LIN {X 0,Y 353.361,Z 397.331,A -85,B 0,C 180,E1 -13405.436,E2 -13405.436} C_VEL
LIN {X 0,Y 353.277,Z 398.793,A -85,B 0,C 180,E1 -13406.578,E2 -13406.578} C_VEL
LIN {X 0,Y 353.318,Z 399.819,A -85,B 0,C 180,E1 -13407.719,E2 -13407.719} C_VEL
LIN {X 0,Y 353.397,Z 400.451,A -85,B 0,C 180,E1 -13408.86,E2 -13408.86} C_VEL
LIN {X 0,Y 353.406,Z 400.682,A -85,B 0,C 180,E1 -13409.999,E2 -13409.999} C_VEL
LIN {X 0,Y 353.397,Z 400.492,A -85,B 0,C 180,E1 -13411.139,E2 -13411.139} C_VEL
LIN {X 0,Y 353.319,Z 399.871,A -85,B 0,C 180,E1 -13412.279,E2 -13412.279} C_VEL
LIN {X 0,Y 353.359,Z 397.445,A -85,B 0,C 180,E1 -13414.562,E2 -13414.562} C_VEL
LIN {X 0,Y 353.439,Z 394.728,A -85,B 0,C 180,E1 -13416.149,E2 -13416.149} C_VEL
LIN {X 0,Y 353.657,Z 390.472,A -85,B 0,C 180,E1 -13417.995,E2 -13417.995} C_VEL
LIN {X 0,Y 354.202,Z 384.355,A -85,B 0,C 180,E1 -13419.997,E2 -13419.997} C_VEL
LIN {X 0,Y 354.848,Z 377.661,A -85,B 0,C 180,E1 -13421.712,E2 -13421.712} C_VEL
LIN {X 0,Y 355.833,Z 369.395,A -85,B 0,C 180,E1 -13423.418,E2 -13423.418} C_VEL
LIN {X 0,Y 356.776,Z 360.995,A -85,B 0,C 180,E1 -13424.837,E2 -13424.837} C_VEL
LIN {X 0,Y 357.808,Z 350.724,A -85,B 0,C 180,E1 -13426.253,E2 -13426.253} C_VEL
LIN {X 0,Y 359.128,Z 339.216,A -85,B 0,C 180,E1 -13427.51,E2 -13427.51} C_VEL
LIN {X 0,Y 359.906,Z 331.464,A -85,B 0,C 180,E1 -13428.205,E2 -13428.205} C_VEL
LIN {X 0,Y 358.662,Z 318.046,A -85,B 0,C 180,E1 -13429.294,E2 -13429.294} C_VEL
LIN {X 0,Y 357.078,Z 305.317,A -85,B 0,C 180,E1 -13430.105,E2 -13430.105} C_VEL
LIN {X 0,Y 354.409,Z 291.71,A -85,B 0,C 180,E1 -13430.818,E2 -13430.818} C_VEL
LIN {X 0,Y 354.987,Z 283.892,A -85,B 0,C 180,E1 -13434.566,E2 -13434.566} C_VEL
LIN {X 0,Y 355.743,Z 276.367,A -85,B 0,C 180,E1 -13438.302,E2 -13438.302} C_VEL
LIN {X 0,Y 356.393,Z 270.304,A -85,B 0,C 180,E1 -13441.447,E2 -13441.447} C_VEL
LIN {X 0,Y 357.263,Z 264.127,A -85,B 0,C 180,E1 -13444.783,E2 -13444.783} C_VEL
LIN {X 0,Y 357.549,Z 260.512,A -85,B 0,C 180,E1 -13446.86,E2 -13446.86} C_VEL
LIN {X 0,Y 357.149,Z 257.096,A -85,B 0,C 180,E1 -13449.027,E2 -13449.027} C_VEL
LIN {X 0,Y 356.306,Z 252.564,A -85,B 0,C 180,E1 -13452.115,E2 -13452.115} C_VEL
LIN {X 0,Y 355.547,Z 248.244,A -85,B 0,C 180,E1 -13455.364,E2 -13455.364} C_VEL
LIN {X 0,Y 354.843,Z 244.322,A -85,B 0,C 180,E1 -13458.686,E2 -13458.686} C_VEL
LIN {X 0,Y 354.814,Z 244.292,A -85,B 0,C 180,E1 -13462.4,E2 -13462.4} C_VEL
LIN {X 0,Y 354.813,Z 244.289,A -85,B 0,C 180,E1 -13464.939,E2 -13464.939} C_VEL
LIN {X 0,Y 354.793,Z 244.291,A -85,B 0,C 180,E1 -13468.403,E2 -13468.403} C_VEL
LIN {X 0,Y 354.849,Z 244.285,A -85,B 0,C 180,E1 -13471.617,E2 -13471.617} C_VEL
LIN {X 0,Y 354.899,Z 244.28,A -85,B 0,C 180,E1 -13474.171,E2 -13474.171} C_VEL
LIN {X 0,Y 354.834,Z 244.284,A -85,B 0,C 180,E1 -13477.892,E2 -13477.892} C_VEL
LIN {X 0,Y 354.922,Z 244.272,A -85,B 0,C 180,E1 -13481.89,E2 -13481.89} C_VEL
LIN {X 0,Y 354.941,Z 244.274,A -85,B 0,C 180,E1 -13485.979,E2 -13485.979} C_VEL
LIN {X 0,Y 354.975,Z 244.268,A -85,B 0,C 180,E1 -13489.734,E2 -13489.734} C_VEL
LIN {X 0,Y 355.111,Z 244.251,A -85,B 0,C 180,E1 -13492.035,E2 -13492.035} C_VEL
LIN {X 0,Y 355.09,Z 244.255,A -85,B 0,C 180,E1 -13494.319,E2 -13494.319} C_VEL
LIN {X 0,Y 355.242,Z 244.233,A -85,B 0,C 180,E1 -13497.731,E2 -13497.731} C_VEL
LIN {X 0,Y 355.395,Z 244.216,A -85,B 0,C 180,E1 -13499.998,E2 -13499.998} C_VEL
LIN {X 0,Y 355.241,Z 244.237,A -85,B 0,C 180,E1 -13502.266,E2 -13502.266} C_VEL
LIN {X 0,Y 355.134,Z 244.251,A -85,B 0,C 180,E1 -13506.817,E2 -13506.817} C_VEL
LIN {X 0,Y 354.999,Z 244.267,A -85,B 0,C 180,E1 -13509.111,E2 -13509.111} C_VEL
LIN {X 0,Y 354.849,Z 244.536,A -85,B 0,C 180,E1 -13511.421,E2 -13511.421} C_VEL
LIN {X 0,Y 354.814,Z 246.447,A -85,B 0,C 180,E1 -13513.938,E2 -13513.938} C_VEL
LIN {X 0,Y 354.579,Z 249.631,A -85,B 0,C 180,E1 -13517.94,E2 -13517.94} C_VEL
LIN {X 0,Y 354.357,Z 252.351,A -85,B 0,C 180,E1 -13521.229,E2 -13521.229} C_VEL
LIN {X 0,Y 354.214,Z 255.232,A -85,B 0,C 180,E1 -13524.622,E2 -13524.622} C_VEL
LIN {X 0,Y 354.178,Z 256.697,A -85,B 0,C 180,E1 -13526.277,E2 -13526.277} C_VEL
LIN {X 0,Y 358.421,Z 270.256,A -85,B 0,C 180,E1 -13527.172,E2 -13527.172} C_VEL
LIN {X 0,Y 361.22,Z 281.692,A -85,B 0,C 180,E1 -13528.071,E2 -13528.071} C_VEL
LIN {X 0,Y 361.763,Z 284.829,A -85,B 0,C 180,E1 -13528.34,E2 -13528.34} C_VEL
LIN {X 0,Y 360.778,Z 296.521,A -85,B 0,C 180,E1 -13529.301,E2 -13529.301} C_VEL
LIN {X 0,Y 359.767,Z 306.717,A -85,B 0,C 180,E1 -13530.359,E2 -13530.359} C_VEL
LIN {X 0,Y 358.53,Z 317.659,A -85,B 0,C 180,E1 -13531.788,E2 -13531.788} C_VEL
LIN {X 0,Y 357.331,Z 327.575,A -85,B 0,C 180,E1 -13533.413,E2 -13533.413} C_VEL
LIN {X 0,Y 356.279,Z 335.9,A -85,B 0,C 180,E1 -13535.138,E2 -13535.138} C_VEL
LIN {X 0,Y 355.322,Z 343.05,A -85,B 0,C 180,E1 -13537.002,E2 -13537.002} C_VEL
LIN {X 0,Y 354.684,Z 347.883,A -85,B 0,C 180,E1 -13538.603,E2 -13538.603} C_VEL
LIN {X 0,Y 354.224,Z 351.564,A -85,B 0,C 180,E1 -13540.149,E2 -13540.149} C_VEL
LIN {X 0,Y 353.897,Z 354.416,A -85,B 0,C 180,E1 -13541.713,E2 -13541.713} C_VEL
LIN {X 0,Y 353.712,Z 355.764,A -85,B 0,C 180,E1 -13542.68,E2 -13542.68} C_VEL
LIN {X 0,Y 353.482,Z 357.354,A -85,B 0,C 180,E1 -13544.296,E2 -13544.296} C_VEL
LIN {X 0,Y 353.306,Z 358.133,A -85,B 0,C 180,E1 -13545.876,E2 -13545.876} C_VEL
LIN {X 0,Y 353.236,Z 358.111,A -85,B 0,C 180,E1 -13547.433,E2 -13547.433} C_VEL
LIN {X 0,Y 353.343,Z 357.276,A -85,B 0,C 180,E1 -13549.093,E2 -13549.093} C_VEL
LIN {X 0,Y 353.518,Z 355.488,A -85,B 0,C 180,E1 -13550.83,E2 -13550.83} C_VEL
LIN {X 0,Y 353.811,Z 352.642,A -85,B 0,C 180,E1 -13552.608,E2 -13552.608} C_VEL
LIN {X 0,Y 354.233,Z 348.577,A -85,B 0,C 180,E1 -13554.429,E2 -13554.429} C_VEL
LIN {X 0,Y 354.798,Z 343.019,A -85,B 0,C 180,E1 -13556.315,E2 -13556.315} C_VEL
LIN {X 0,Y 355.556,Z 335.815,A -85,B 0,C 180,E1 -13558.201,E2 -13558.201} C_VEL
LIN {X 0,Y 356.447,Z 327.335,A -85,B 0,C 180,E1 -13559.958,E2 -13559.958} C_VEL
LIN {X 0,Y 357.46,Z 317.879,A -85,B 0,C 180,E1 -13561.526,E2 -13561.526} C_VEL
LIN {X 0,Y 358.429,Z 307.732,A -85,B 0,C 180,E1 -13562.879,E2 -13562.879} C_VEL
LIN {X 0,Y 359.445,Z 296.584,A -85,B 0,C 180,E1 -13564.074,E2 -13564.074} C_VEL
LIN {X 0,Y 360.348,Z 284.915,A -85,B 0,C 180,E1 -13565.055,E2 -13565.055} C_VEL
LIN {X 0,Y 360.523,Z 282.568,A -85,B 0,C 180,E1 -13565.222,E2 -13565.222} C_VEL
LIN {X 0,Y 358.332,Z 271.377,A -85,B 0,C 180,E1 -13566.056,E2 -13566.056} C_VEL
LIN {X 0,Y 354.955,Z 258.671,A -85,B 0,C 180,E1 -13566.827,E2 -13566.827} C_VEL
LIN {X 0,Y 353.815,Z 254.351,A -85,B 0,C 180,E1 -13567.057,E2 -13567.057} C_VEL
LIN {X 0,Y 353.884,Z 251.226,A -85,B 0,C 180,E1 -13570.269,E2 -13570.269} C_VEL
LIN {X 0,Y 354.007,Z 248.917,A -85,B 0,C 180,E1 -13572.676,E2 -13572.676} C_VEL
LIN {X 0,Y 354.162,Z 245.343,A -85,B 0,C 180,E1 -13576.485,E2 -13576.485} C_VEL
LIN {X 0,Y 354.227,Z 244.505,A -85,B 0,C 180,E1 -13577.395,E2 -13577.395} C_VEL
LIN {X 0,Y 354.713,Z 244.299,A -85,B 0,C 180,E1 -13580.881,E2 -13580.881} C_VEL
LIN {X 0,Y 355.055,Z 244.259,A -85,B 0,C 180,E1 -13583.18,E2 -13583.18} C_VEL
LIN {X 0,Y 355.231,Z 244.236,A -85,B 0,C 180,E1 -13587.733,E2 -13587.733} C_VEL
LIN {X 0,Y 355.383,Z 244.215,A -85,B 0,C 180,E1 -13590.001,E2 -13590.001} C_VEL
LIN {X 0,Y 355.231,Z 244.233,A -85,B 0,C 180,E1 -13592.268,E2 -13592.268} C_VEL
LIN {X 0,Y 355.123,Z 244.249,A -85,B 0,C 180,E1 -13596.82,E2 -13596.82} C_VEL
LIN {X 0,Y 355.002,Z 244.267,A -85,B 0,C 180,E1 -13599.113,E2 -13599.113} C_VEL
LIN {X 0,Y 354.911,Z 244.275,A -85,B 0,C 180,E1 -13602.582,E2 -13602.582} C_VEL
LIN {X 0,Y 354.875,Z 244.278,A -85,B 0,C 180,E1 -13606.097,E2 -13606.097} C_VEL
LIN {X 0,Y 354.896,Z 244.276,A -85,B 0,C 180,E1 -13608.473,E2 -13608.473} C_VEL
LIN {X 0,Y 354.874,Z 244.278,A -85,B 0,C 180,E1 -13612.104,E2 -13612.104} C_VEL
LIN {X 0,Y 354.887,Z 244.276,A -85,B 0,C 180,E1 -13615.829,E2 -13615.829} C_VEL
LIN {X 0,Y 354.841,Z 244.282,A -85,B 0,C 180,E1 -13619.68,E2 -13619.68} C_VEL
LIN {X 0,Y 354.795,Z 244.288,A -85,B 0,C 180,E1 -13623.704,E2 -13623.704} C_VEL
LIN {X 0,Y 354.789,Z 244.292,A -85,B 0,C 180,E1 -13626.461,E2 -13626.461} C_VEL
LIN {X 0,Y 354.814,Z 244.285,A -85,B 0,C 180,E1 -13629.426,E2 -13629.426} C_VEL
LIN {X 0,Y 354.826,Z 244.284,A -85,B 0,C 180,E1 -13631.226,E2 -13631.226} C_VEL
LIN {X 0,Y 354.125,Z 244.375,A -85,B 0,C 180,E1 -13632.173,E2 -13632.173} C_VEL
LIN {X 0,Y 351.255,Z 244.729,A -85,B 0,C 180,E1 -13633.712,E2 -13633.712} C_VEL
LIN {X 0,Y 348.861,Z 245.029,A -85,B 0,C 180,E1 -13634.957,E2 -13634.957} C_VEL
LIN {X 0,Y 347.859,Z 245.152,A -85,B 0,C 180,E1 -13635.921,E2 -13635.921} C_VEL
LIN {X 0,Y 347.79,Z 245.161,A -85,B 0,C 180,E1 -13636.247,E2 -13636.247} C_VEL
LIN {X 0,Y 347.778,Z 245.165,A -85,B 0,C 180,E1 -13640.168,E2 -13640.168} C_VEL
LIN {X 0,Y 347.783,Z 245.165,A -85,B 0,C 180,E1 -13644.127,E2 -13644.127} C_VEL
LIN {X 0,Y 347.759,Z 245.169,A -85,B 0,C 180,E1 -13648.305,E2 -13648.305} C_VEL
LIN {X 0,Y 347.802,Z 245.159,A -85,B 0,C 180,E1 -13650.992,E2 -13650.992} C_VEL
LIN {X 0,Y 347.828,Z 245.156,A -85,B 0,C 180,E1 -13653.61,E2 -13653.61} C_VEL
LIN {X 0,Y 347.786,Z 245.166,A -85,B 0,C 180,E1 -13656.164,E2 -13656.164} C_VEL
LIN {X 0,Y 347.816,Z 245.161,A -85,B 0,C 180,E1 -13659.912,E2 -13659.912} C_VEL
LIN {X 0,Y 347.865,Z 245.154,A -85,B 0,C 180,E1 -13662.362,E2 -13662.362} C_VEL
LIN {X 0,Y 347.897,Z 245.152,A -85,B 0,C 180,E1 -13665.973,E2 -13665.973} C_VEL
LIN {X 0,Y 347.927,Z 245.145,A -85,B 0,C 180,E1 -13669.528,E2 -13669.528} C_VEL
LIN {X 0,Y 348.08,Z 245.124,A -85,B 0,C 180,E1 -13673.044,E2 -13673.044} C_VEL
LIN {X 0,Y 348.208,Z 245.113,A -85,B 0,C 180,E1 -13677.689,E2 -13677.689} C_VEL
LIN {X 0,Y 348.347,Z 245.094,A -85,B 0,C 180,E1 -13680.002,E2 -13680.002} C_VEL
LIN {X 0,Y 348.208,Z 245.109,A -85,B 0,C 180,E1 -13682.315,E2 -13682.315} C_VEL
LIN {X 0,Y 348.067,Z 245.126,A -85,B 0,C 180,E1 -13686.96,E2 -13686.96} C_VEL
LIN {X 0,Y 347.901,Z 245.146,A -85,B 0,C 180,E1 -13690.477,E2 -13690.477} C_VEL
LIN {X 0,Y 347.904,Z 245.147,A -85,B 0,C 180,E1 -13694.151,E2 -13694.151} C_VEL
LIN {X 0,Y 347.897,Z 245.147,A -85,B 0,C 180,E1 -13698.291,E2 -13698.291} C_VEL
LIN {X 0,Y 347.793,Z 245.163,A -85,B 0,C 180,E1 -13701.636,E2 -13701.636} C_VEL
LIN {X 0,Y 347.818,Z 245.16,A -85,B 0,C 180,E1 -13705.11,E2 -13705.11} C_VEL
LIN {X 0,Y 347.815,Z 245.159,A -85,B 0,C 180,E1 -13707.695,E2 -13707.695} C_VEL
LIN {X 0,Y 347.756,Z 245.164,A -85,B 0,C 180,E1 -13710.349,E2 -13710.349} C_VEL
LIN {X 0,Y 347.755,Z 245.164,A -85,B 0,C 180,E1 -13714.045,E2 -13714.045} C_VEL
LIN {X 0,Y 347.768,Z 245.167,A -85,B 0,C 180,E1 -13717.322,E2 -13717.322} C_VEL
LIN {X 0,Y 347.739,Z 245.169,A -85,B 0,C 180,E1 -13720.298,E2 -13720.298} C_VEL
LIN {X 0,Y 347.776,Z 245.188,A -85,B 0,C 180,E1 -13723.096,E2 -13723.096} C_VEL
LIN {X 0,Y 348.766,Z 250.707,A -85,B 0,C 180,E1 -13726.753,E2 -13726.753} C_VEL
LIN {X 0,Y 349.769,Z 255.89,A -85,B 0,C 180,E1 -13729.985,E2 -13729.985} C_VEL
LIN {X 0,Y 350.482,Z 261.02,A -85,B 0,C 180,E1 -13733.017,E2 -13733.017} C_VEL
LIN {X 0,Y 350.039,Z 266.11,A -85,B 0,C 180,E1 -13735.793,E2 -13735.793} C_VEL
LIN {X 0,Y 349.258,Z 272.455,A -85,B 0,C 180,E1 -13739.127,E2 -13739.127} C_VEL
LIN {X 0,Y 348.563,Z 279.107,A -85,B 0,C 180,E1 -13742.521,E2 -13742.521} C_VEL
LIN {X 0,Y 347.849,Z 286.426,A -85,B 0,C 180,E1 -13746.166,E2 -13746.166} C_VEL
LIN {X 0,Y 347.374,Z 292.917,A -85,B 0,C 180,E1 -13749.291,E2 -13749.291} C_VEL
LIN {X 0,Y 349.68,Z 306.543,A -85,B 0,C 180,E1 -13749.923,E2 -13749.923} C_VEL
LIN {X 0,Y 351.362,Z 319.394,A -85,B 0,C 180,E1 -13750.738,E2 -13750.738} C_VEL
LIN {X 0,Y 352.641,Z 331.31,A -85,B 0,C 180,E1 -13751.706,E2 -13751.706} C_VEL
LIN {X 0,Y 351.608,Z 342.057,A -85,B 0,C 180,E1 -13752.702,E2 -13752.702} C_VEL
LIN {X 0,Y 350.415,Z 353.068,A -85,B 0,C 180,E1 -13753.988,E2 -13753.988} C_VEL
LIN {X 0,Y 349.438,Z 362.972,A -85,B 0,C 180,E1 -13755.439,E2 -13755.439} C_VEL
LIN {X 0,Y 348.513,Z 371.083,A -85,B 0,C 180,E1 -13756.887,E2 -13756.887} C_VEL
LIN {X 0,Y 347.547,Z 379.047,A -85,B 0,C 180,E1 -13758.628,E2 -13758.628} C_VEL
LIN {X 0,Y 347.062,Z 384.449,A -85,B 0,C 180,E1 -13760.088,E2 -13760.088} C_VEL
LIN {X 0,Y 346.596,Z 389.732,A -85,B 0,C 180,E1 -13761.839,E2 -13761.839} C_VEL
LIN {X 0,Y 346.342,Z 394.426,A -85,B 0,C 180,E1 -13763.896,E2 -13763.896} C_VEL
LIN {X 0,Y 346.276,Z 396.866,A -85,B 0,C 180,E1 -13765.343,E2 -13765.343} C_VEL
LIN {X 0,Y 346.201,Z 398.344,A -85,B 0,C 180,E1 -13766.508,E2 -13766.508} C_VEL
LIN {X 0,Y 346.317,Z 400.016,A -85,B 0,C 180,E1 -13768.837,E2 -13768.837} C_VEL
LIN {X 0,Y 346.345,Z 400.255,A -85,B 0,C 180,E1 -13769.999,E2 -13769.999} C_VEL
LIN {X 0,Y 346.318,Z 400.077,A -85,B 0,C 180,E1 -13771.162,E2 -13771.162} C_VEL
LIN {X 0,Y 346.207,Z 398.452,A -85,B 0,C 180,E1 -13773.491,E2 -13773.491} C_VEL
LIN {X 0,Y 346.273,Z 397.045,A -85,B 0,C 180,E1 -13774.656,E2 -13774.656} C_VEL
LIN {X 0,Y 346.335,Z 394.684,A -85,B 0,C 180,E1 -13776.092,E2 -13776.092} C_VEL
LIN {X 0,Y 346.595,Z 390.1,A -85,B 0,C 180,E1 -13778.159,E2 -13778.159} C_VEL
LIN {X 0,Y 347.072,Z 384.988,A -85,B 0,C 180,E1 -13779.91,E2 -13779.91} C_VEL
LIN {X 0,Y 347.687,Z 378.594,A -85,B 0,C 180,E1 -13781.661,E2 -13781.661} C_VEL
LIN {X 0,Y 348.717,Z 370.636,A -85,B 0,C 180,E1 -13783.401,E2 -13783.401} C_VEL
LIN {X 0,Y 349.88,Z 360.769,A -85,B 0,C 180,E1 -13785.136,E2 -13785.136} C_VEL
LIN {X 0,Y 350.976,Z 350.569,A -85,B 0,C 180,E1 -13786.579,E2 -13786.579} C_VEL
LIN {X 0,Y 352.371,Z 339.126,A -85,B 0,C 180,E1 -13787.857,E2 -13787.857} C_VEL
LIN {X 0,Y 353.017,Z 331.463,A -85,B 0,C 180,E1 -13788.574,E2 -13788.574} C_VEL
LIN {X 0,Y 351.865,Z 318.429,A -85,B 0,C 180,E1 -13789.665,E2 -13789.665} C_VEL
LIN {X 0,Y 350.342,Z 305.957,A -85,B 0,C 180,E1 -13790.504,E2 -13790.504} C_VEL
LIN {X 0,Y 347.884,Z 293.833,A -85,B 0,C 180,E1 -13791.177,E2 -13791.177} C_VEL
LIN {X 0,Y 347.426,Z 291.28,A -85,B 0,C 180,E1 -13791.298,E2 -13791.298} C_VEL
LIN {X 0,Y 348.044,Z 283.59,A -85,B 0,C 180,E1 -13795.09,E2 -13795.09} C_VEL
LIN {X 0,Y 348.821,Z 276.111,A -85,B 0,C 180,E1 -13798.917,E2 -13798.917} C_VEL
LIN {X 0,Y 349.564,Z 269.643,A -85,B 0,C 180,E1 -13802.389,E2 -13802.389} C_VEL
LIN {X 0,Y 350.429,Z 263.99,A -85,B 0,C 180,E1 -13805.563,E2 -13805.563} C_VEL
LIN {X 0,Y 350.493,Z 260.48,A -85,B 0,C 180,E1 -13807.703,E2 -13807.703} C_VEL
LIN {X 0,Y 349.865,Z 256.648,A -85,B 0,C 180,E1 -13810.239,E2 -13810.239} C_VEL
LIN {X 0,Y 349.01,Z 252.127,A -85,B 0,C 180,E1 -13813.535,E2 -13813.535} C_VEL
LIN {X 0,Y 348.364,Z 248.203,A -85,B 0,C 180,E1 -13816.69,E2 -13816.69} C_VEL
LIN {X 0,Y 347.784,Z 245.166,A -85,B 0,C 180,E1 -13819.537,E2 -13819.537} C_VEL
LIN {X 0,Y 347.768,Z 245.169,A -85,B 0,C 180,E1 -13822.678,E2 -13822.678} C_VEL
LIN {X 0,Y 347.749,Z 245.172,A -85,B 0,C 180,E1 -13825.955,E2 -13825.955} C_VEL
LIN {X 0,Y 347.764,Z 245.168,A -85,B 0,C 180,E1 -13829.652,E2 -13829.652} C_VEL
LIN {X 0,Y 347.851,Z 245.157,A -85,B 0,C 180,E1 -13832.743,E2 -13832.743} C_VEL
LIN {X 0,Y 347.788,Z 245.164,A -85,B 0,C 180,E1 -13836.16,E2 -13836.16} C_VEL
LIN {X 0,Y 347.816,Z 245.156,A -85,B 0,C 180,E1 -13839.908,E2 -13839.908} C_VEL
LIN {X 0,Y 347.865,Z 245.15,A -85,B 0,C 180,E1 -13842.357,E2 -13842.357} C_VEL
LIN {X 0,Y 347.895,Z 245.151,A -85,B 0,C 180,E1 -13845.969,E2 -13845.969} C_VEL
LIN {X 0,Y 347.926,Z 245.145,A -85,B 0,C 180,E1 -13849.524,E2 -13849.524} C_VEL
LIN {X 0,Y 348.071,Z 245.127,A -85,B 0,C 180,E1 -13851.873,E2 -13851.873} C_VEL
LIN {X 0,Y 348.065,Z 245.129,A -85,B 0,C 180,E1 -13854.204,E2 -13854.204} C_VEL
LIN {X 0,Y 348.205,Z 245.11,A -85,B 0,C 180,E1 -13857.685,E2 -13857.685} C_VEL
LIN {X 0,Y 348.365,Z 245.092,A -85,B 0,C 180,E1 -13859.998,E2 -13859.998} C_VEL
LIN {X 0,Y 348.203,Z 245.113,A -85,B 0,C 180,E1 -13862.312,E2 -13862.312} C_VEL
LIN {X 0,Y 348.103,Z 245.127,A -85,B 0,C 180,E1 -13866.956,E2 -13866.956} C_VEL
LIN {X 0,Y 347.931,Z 245.148,A -85,B 0,C 180,E1 -13869.297,E2 -13869.297} C_VEL
LIN {X 0,Y 347.849,Z 245.161,A -85,B 0,C 180,E1 -13870.475,E2 -13870.475} C_VEL
LIN {X 0,Y 347.784,Z 247.675,A -85,B 0,C 180,E1 -13874.078,E2 -13874.078} C_VEL
LIN {X 0,Y 347.574,Z 250.449,A -85,B 0,C 180,E1 -13877.654,E2 -13877.654} C_VEL
LIN {X 0,Y 347.335,Z 253.534,A -85,B 0,C 180,E1 -13881.448,E2 -13881.448} C_VEL
LIN {X 0,Y 347.139,Z 256.657,A -85,B 0,C 180,E1 -13885.158,E2 -13885.158} C_VEL
LIN {X 0,Y 347.121,Z 257.163,A -85,B 0,C 180,E1 -13885.762,E2 -13885.762} C_VEL
LIN {X 0,Y 351.833,Z 271.894,A -85,B 0,C 180,E1 -13886.796,E2 -13886.796} C_VEL
LIN {X 0,Y 354.664,Z 283.756,A -85,B 0,C 180,E1 -13887.783,E2 -13887.783} C_VEL
LIN {X 0,Y 355.097,Z 285.746,A -85,B 0,C 180,E1 -13887.97,E2 -13887.97} C_VEL
LIN {X 0,Y 354.11,Z 297.116,A -85,B 0,C 180,E1 -13888.928,E2 -13888.928} C_VEL
LIN {X 0,Y 352.84,Z 308.832,A -85,B 0,C 180,E1 -13890.192,E2 -13890.192} C_VEL
LIN {X 0,Y 351.623,Z 319.419,A -85,B 0,C 180,E1 -13891.643,E2 -13891.643} C_VEL
LIN {X 0,Y 350.492,Z 328.125,A -85,B 0,C 180,E1 -13893.118,E2 -13893.118} C_VEL
LIN {X 0,Y 349.479,Z 335.78,A -85,B 0,C 180,E1 -13894.723,E2 -13894.723} C_VEL
LIN {X 0,Y 348.394,Z 343.338,A -85,B 0,C 180,E1 -13896.715,E2 -13896.715} C_VEL
LIN {X 0,Y 347.726,Z 348.23,A -85,B 0,C 180,E1 -13898.361,E2 -13898.361} C_VEL
LIN {X 0,Y 347.116,Z 352.84,A -85,B 0,C 180,E1 -13900.38,E2 -13900.38} C_VEL
LIN {X 0,Y 346.766,Z 355.458,A -85,B 0,C 180,E1 -13901.973,E2 -13901.973} C_VEL
LIN {X 0,Y 346.484,Z 357.303,A -85,B 0,C 180,E1 -13903.599,E2 -13903.599} C_VEL
LIN {X 0,Y 346.277,Z 358.373,A -85,B 0,C 180,E1 -13905.26,E2 -13905.26} C_VEL
LIN {X 0,Y 346.165,Z 358.629,A -85,B 0,C 180,E1 -13906.957,E2 -13906.957} C_VEL
LIN {X 0,Y 346.215,Z 358.016,A -85,B 0,C 180,E1 -13908.68,E2 -13908.68} C_VEL
LIN {X 0,Y 346.383,Z 356.463,A -85,B 0,C 180,E1 -13910.44,E2 -13910.44} C_VEL
LIN {X 0,Y 346.743,Z 353.31,A -85,B 0,C 180,E1 -13912.552,E2 -13912.552} C_VEL
LIN {X 0,Y 347.058,Z 350.115,A -85,B 0,C 180,E1 -13914.092,E2 -13914.092} C_VEL
LIN {X 0,Y 347.617,Z 344.953,A -85,B 0,C 180,E1 -13915.984,E2 -13915.984} C_VEL
LIN {X 0,Y 348.319,Z 338.108,A -85,B 0,C 180,E1 -13917.928,E2 -13917.928} C_VEL
LIN {X 0,Y 349.101,Z 331.426,A -85,B 0,C 180,E1 -13919.449,E2 -13919.449} C_VEL
LIN {X 0,Y 350.076,Z 322.94,A -85,B 0,C 180,E1 -13921.033,E2 -13921.033} C_VEL
LIN {X 0,Y 351.14,Z 312.518,A -85,B 0,C 180,E1 -13922.592,E2 -13922.592} C_VEL
LIN {X 0,Y 352.253,Z 301.01,A -85,B 0,C 180,E1 -13923.965,E2 -13923.965} C_VEL
LIN {X 0,Y 353.249,Z 289.115,A -85,B 0,C 180,E1 -13925.069,E2 -13925.069} C_VEL
LIN {X 0,Y 353.691,Z 283.577,A -85,B 0,C 180,E1 -13925.494,E2 -13925.494} C_VEL
LIN {X 0,Y 351.235,Z 271.767,A -85,B 0,C 180,E1 -13926.411,E2 -13926.411} C_VEL
LIN {X 0,Y 347.924,Z 259.115,A -85,B 0,C 180,E1 -13927.197,E2 -13927.197} C_VEL
LIN {X 0,Y 346.766,Z 254.748,A -85,B 0,C 180,E1 -13927.431,E2 -13927.431} C_VEL
LIN {X 0,Y 346.872,Z 251.238,A -85,B 0,C 180,E1 -13931.085,E2 -13931.085} C_VEL
LIN {X 0,Y 346.945,Z 248.94,A -85,B 0,C 180,E1 -13933.526,E2 -13933.526} C_VEL
LIN {X 0,Y 347.173,Z 245.603,A -85,B 0,C 180,E1 -13937.134,E2 -13937.134} C_VEL
LIN {X 0,Y 347.46,Z 245.207,A -85,B 0,C 180,E1 -13939.512,E2 -13939.512} C_VEL
LIN {X 0,Y 348.013,Z 245.135,A -85,B 0,C 180,E1 -13943.041,E2 -13943.041} C_VEL
LIN {X 0,Y 348.193,Z 245.112,A -85,B 0,C 180,E1 -13947.687,E2 -13947.687} C_VEL
LIN {X 0,Y 348.353,Z 245.09,A -85,B 0,C 180,E1 -13950.001,E2 -13950.001} C_VEL
LIN {X 0,Y 348.193,Z 245.11,A -85,B 0,C 180,E1 -13952.314,E2 -13952.314} C_VEL
LIN {X 0,Y 348.091,Z 245.127,A -85,B 0,C 180,E1 -13956.959,E2 -13956.959} C_VEL
LIN {X 0,Y 347.954,Z 245.144,A -85,B 0,C 180,E1 -13959.299,E2 -13959.299} C_VEL
LIN {X 0,Y 347.879,Z 245.153,A -85,B 0,C 180,E1 -13962.84,E2 -13962.84} C_VEL
LIN {X 0,Y 347.825,Z 245.157,A -85,B 0,C 180,E1 -13966.433,E2 -13966.433} C_VEL
LIN {X 0,Y 347.849,Z 245.158,A -85,B 0,C 180,E1 -13968.861,E2 -13968.861} C_VEL
LIN {X 0,Y 347.795,Z 245.162,A -85,B 0,C 180,E1 -13972.578,E2 -13972.578} C_VEL
LIN {X 0,Y 347.808,Z 245.161,A -85,B 0,C 180,E1 -13975.109,E2 -13975.109} C_VEL
LIN {X 0,Y 347.797,Z 245.159,A -85,B 0,C 180,E1 -13977.696,E2 -13977.696} C_VEL
LIN {X 0,Y 347.752,Z 245.167,A -85,B 0,C 180,E1 -13980.348,E2 -13980.348} C_VEL
LIN {X 0,Y 347.733,Z 245.171,A -85,B 0,C 180,E1 -13984.466,E2 -13984.466} C_VEL
LIN {X 0,Y 347.766,Z 245.164,A -85,B 0,C 180,E1 -13987.991,E2 -13987.991} C_VEL
LIN {X 0,Y 347.775,Z 245.162,A -85,B 0,C 180,E1 -13991.611,E2 -13991.611} C_VEL
LIN {X 0,Y 347.822,Z 245.158,A -85,B 0,C 180,E1 -13995.008,E2 -13995.008} C_VEL
LIN {X 0,Y 347.79,Z 245.161,A -85,B 0,C 180,E1 -13996.247,E2 -13996.247} C_VEL
LIN {X 0,Y 347.143,Z 245.247,A -85,B 0,C 180,E1 -13997.214,E2 -13997.214} C_VEL
LIN {X 0,Y 344.257,Z 245.605,A -85,B 0,C 180,E1 -13998.786,E2 -13998.786} C_VEL
LIN {X 0,Y 341.806,Z 245.908,A -85,B 0,C 180,E1 -14000.059,E2 -14000.059} C_VEL
LIN {X 0,Y 340.774,Z 246.035,A -85,B 0,C 180,E1 -14001.044,E2 -14001.044} C_VEL
LIN {X 0,Y 340.701,Z 246.042,A -85,B 0,C 180,E1 -14001.378,E2 -14001.378} C_VEL
LIN {X 0,Y 340.713,Z 246.044,A -85,B 0,C 180,E1 -14004.724,E2 -14004.724} C_VEL
LIN {X 0,Y 340.711,Z 246.042,A -85,B 0,C 180,E1 -14008.96,E2 -14008.96} C_VEL
LIN {X 0,Y 340.776,Z 246.037,A -85,B 0,C 180,E1 -14012.476,E2 -14012.476} C_VEL
LIN {X 0,Y 340.753,Z 246.038,A -85,B 0,C 180,E1 -14015.641,E2 -14015.641} C_VEL
LIN {X 0,Y 340.746,Z 246.038,A -85,B 0,C 180,E1 -14019.477,E2 -14019.477} C_VEL
LIN {X 0,Y 340.857,Z 246.029,A -85,B 0,C 180,E1 -14021.987,E2 -14021.987} C_VEL
LIN {X 0,Y 340.869,Z 246.025,A -85,B 0,C 180,E1 -14025.707,E2 -14025.707} C_VEL
LIN {X 0,Y 340.87,Z 246.023,A -85,B 0,C 180,E1 -14029.308,E2 -14029.308} C_VEL
LIN {X 0,Y 341.047,Z 246,A -85,B 0,C 180,E1 -14032.9,E2 -14032.9} C_VEL
LIN {X 0,Y 341.17,Z 245.989,A -85,B 0,C 180,E1 -14037.641,E2 -14037.641} C_VEL
LIN {X 0,Y 341.298,Z 245.972,A -85,B 0,C 180,E1 -14040.002,E2 -14040.002} C_VEL
LIN {X 0,Y 341.17,Z 245.985,A -85,B 0,C 180,E1 -14042.363,E2 -14042.363} C_VEL
LIN {X 0,Y 341.013,Z 246.005,A -85,B 0,C 180,E1 -14047.105,E2 -14047.105} C_VEL
LIN {X 0,Y 340.852,Z 246.024,A -85,B 0,C 180,E1 -14050.696,E2 -14050.696} C_VEL
LIN {X 0,Y 340.868,Z 246.022,A -85,B 0,C 180,E1 -14054.326,E2 -14054.326} C_VEL
LIN {X 0,Y 340.843,Z 246.025,A -85,B 0,C 180,E1 -14058.468,E2 -14058.468} C_VEL
LIN {X 0,Y 340.76,Z 246.037,A -85,B 0,C 180,E1 -14061.858,E2 -14061.858} C_VEL
LIN {X 0,Y 340.778,Z 246.036,A -85,B 0,C 180,E1 -14065.666,E2 -14065.666} C_VEL
LIN {X 0,Y 340.735,Z 246.039,A -85,B 0,C 180,E1 -14068.322,E2 -14068.322} C_VEL
LIN {X 0,Y 340.705,Z 246.046,A -85,B 0,C 180,E1 -14071.046,E2 -14071.046} C_VEL
LIN {X 0,Y 340.725,Z 246.045,A -85,B 0,C 180,E1 -14075.28,E2 -14075.28} C_VEL
LIN {X 0,Y 340.717,Z 246.045,A -85,B 0,C 180,E1 -14078.387,E2 -14078.387} C_VEL
LIN {X 0,Y 340.732,Z 246.04,A -85,B 0,C 180,E1 -14082.421,E2 -14082.421} C_VEL
LIN {X 0,Y 340.77,Z 246.34,A -85,B 0,C 180,E1 -14082.891,E2 -14082.891} C_VEL
LIN {X 0,Y 341.624,Z 250.986,A -85,B 0,C 180,E1 -14086.059,E2 -14086.059} C_VEL
LIN {X 0,Y 342.6,Z 256.138,A -85,B 0,C 180,E1 -14089.379,E2 -14089.379} C_VEL
LIN {X 0,Y 343.312,Z 260.621,A -85,B 0,C 180,E1 -14092.11,E2 -14092.11} C_VEL
LIN {X 0,Y 343.413,Z 263.171,A -85,B 0,C 180,E1 -14093.594,E2 -14093.594} C_VEL
LIN {X 0,Y 342.894,Z 268.273,A -85,B 0,C 180,E1 -14096.399,E2 -14096.399} C_VEL
LIN {X 0,Y 342.091,Z 274.323,A -85,B 0,C 180,E1 -14099.641,E2 -14099.641} C_VEL
LIN {X 0,Y 341.365,Z 280.939,A -85,B 0,C 180,E1 -14103.067,E2 -14103.067} C_VEL
LIN {X 0,Y 340.761,Z 287.25,A -85,B 0,C 180,E1 -14106.285,E2 -14106.285} C_VEL
LIN {X 0,Y 340.357,Z 292.422,A -85,B 0,C 180,E1 -14108.866,E2 -14108.866} C_VEL
LIN {X 0,Y 342.895,Z 307.742,A -85,B 0,C 180,E1 -14109.635,E2 -14109.635} C_VEL
LIN {X 0,Y 344.454,Z 319.682,A -85,B 0,C 180,E1 -14110.43,E2 -14110.43} C_VEL
LIN {X 0,Y 345.729,Z 332.17,A -85,B 0,C 180,E1 -14111.48,E2 -14111.48} C_VEL
LIN {X 0,Y 344.484,Z 343.953,A -85,B 0,C 180,E1 -14112.64,E2 -14112.64} C_VEL
LIN {X 0,Y 343.316,Z 354.54,A -85,B 0,C 180,E1 -14113.957,E2 -14113.957} C_VEL
LIN {X 0,Y 342.312,Z 364.116,A -85,B 0,C 180,E1 -14115.433,E2 -14115.433} C_VEL
LIN {X 0,Y 341.169,Z 373.336,A -85,B 0,C 180,E1 -14117.205,E2 -14117.205} C_VEL
LIN {X 0,Y 340.329,Z 380.762,A -85,B 0,C 180,E1 -14118.987,E2 -14118.987} C_VEL
LIN {X 0,Y 339.703,Z 387.596,A -85,B 0,C 180,E1 -14121.073,E2 -14121.073} C_VEL
LIN {X 0,Y 339.353,Z 392.094,A -85,B 0,C 180,E1 -14122.861,E2 -14122.861} C_VEL
LIN {X 0,Y 339.264,Z 394.466,A -85,B 0,C 180,E1 -14124.054,E2 -14124.054} C_VEL
LIN {X 0,Y 339.196,Z 396.398,A -85,B 0,C 180,E1 -14125.245,E2 -14125.245} C_VEL
LIN {X 0,Y 339.126,Z 397.893,A -85,B 0,C 180,E1 -14126.435,E2 -14126.435} C_VEL
LIN {X 0,Y 339.224,Z 399.579,A -85,B 0,C 180,E1 -14128.812,E2 -14128.812} C_VEL
LIN {X 0,Y 339.286,Z 399.828,A -85,B 0,C 180,E1 -14129.999,E2 -14129.999} C_VEL
LIN {X 0,Y 339.224,Z 399.661,A -85,B 0,C 180,E1 -14131.186,E2 -14131.186} C_VEL
LIN {X 0,Y 339.132,Z 398.054,A -85,B 0,C 180,E1 -14133.564,E2 -14133.564} C_VEL
LIN {X 0,Y 339.191,Z 396.656,A -85,B 0,C 180,E1 -14134.753,E2 -14134.753} C_VEL
LIN {X 0,Y 339.282,Z 393.721,A -85,B 0,C 180,E1 -14136.541,E2 -14136.541} C_VEL
LIN {X 0,Y 339.551,Z 389.753,A -85,B 0,C 180,E1 -14138.33,E2 -14138.33} C_VEL
LIN {X 0,Y 340.06,Z 384.661,A -85,B 0,C 180,E1 -14140.117,E2 -14140.117} C_VEL
LIN {X 0,Y 340.696,Z 378.292,A -85,B 0,C 180,E1 -14141.904,E2 -14141.904} C_VEL
LIN {X 0,Y 341.786,Z 370.377,A -85,B 0,C 180,E1 -14143.678,E2 -14143.678} C_VEL
LIN {X 0,Y 342.789,Z 362.338,A -85,B 0,C 180,E1 -14145.153,E2 -14145.153} C_VEL
LIN {X 0,Y 344.007,Z 351.512,A -85,B 0,C 180,E1 -14146.772,E2 -14146.772} C_VEL
LIN {X 0,Y 345.441,Z 340.473,A -85,B 0,C 180,E1 -14148.074,E2 -14148.074} C_VEL
LIN {X 0,Y 346.226,Z 333.086,A -85,B 0,C 180,E1 -14148.798,E2 -14148.798} C_VEL
LIN {X 0,Y 345.334,Z 321.356,A -85,B 0,C 180,E1 -14149.865,E2 -14149.865} C_VEL
LIN {X 0,Y 343.927,Z 308.556,A -85,B 0,C 180,E1 -14150.795,E2 -14150.795} C_VEL
LIN {X 0,Y 341.557,Z 296.168,A -85,B 0,C 180,E1 -14151.542,E2 -14151.542} C_VEL
LIN {X 0,Y 340.383,Z 290.836,A -85,B 0,C 180,E1 -14151.817,E2 -14151.817} C_VEL
LIN {X 0,Y 341.086,Z 283.301,A -85,B 0,C 180,E1 -14155.638,E2 -14155.638} C_VEL
LIN {X 0,Y 341.908,Z 275.877,A -85,B 0,C 180,E1 -14159.558,E2 -14159.558} C_VEL
LIN {X 0,Y 342.605,Z 270.109,A -85,B 0,C 180,E1 -14162.746,E2 -14162.746} C_VEL
LIN {X 0,Y 343.43,Z 265.015,A -85,B 0,C 180,E1 -14165.676,E2 -14165.676} C_VEL
LIN {X 0,Y 343.482,Z 261.526,A -85,B 0,C 180,E1 -14167.866,E2 -14167.866} C_VEL
LIN {X 0,Y 342.7,Z 256.958,A -85,B 0,C 180,E1 -14171.013,E2 -14171.013} C_VEL
LIN {X 0,Y 341.886,Z 252.577,A -85,B 0,C 180,E1 -14174.339,E2 -14174.339} C_VEL
LIN {X 0,Y 341.182,Z 248.472,A -85,B 0,C 180,E1 -14177.863,E2 -14177.863} C_VEL
LIN {X 0,Y 340.713,Z 246.045,A -85,B 0,C 180,E1 -14180.248,E2 -14180.248} C_VEL
LIN {X 0,Y 340.713,Z 246.046,A -85,B 0,C 180,E1 -14183.557,E2 -14183.557} C_VEL
LIN {X 0,Y 340.693,Z 246.05,A -85,B 0,C 180,E1 -14186.152,E2 -14186.152} C_VEL
LIN {X 0,Y 340.775,Z 246.037,A -85,B 0,C 180,E1 -14190.331,E2 -14190.331} C_VEL
LIN {X 0,Y 340.804,Z 246.035,A -85,B 0,C 180,E1 -14193.018,E2 -14193.018} C_VEL
LIN {X 0,Y 340.728,Z 246.042,A -85,B 0,C 180,E1 -14196.925,E2 -14196.925} C_VEL
LIN {X 0,Y 340.793,Z 246.035,A -85,B 0,C 180,E1 -14200.732,E2 -14200.732} C_VEL
LIN {X 0,Y 340.785,Z 246.037,A -85,B 0,C 180,E1 -14203.217,E2 -14203.217} C_VEL
LIN {X 0,Y 340.842,Z 246.026,A -85,B 0,C 180,E1 -14206.889,E2 -14206.889} C_VEL
LIN {X 0,Y 340.926,Z 246.02,A -85,B 0,C 180,E1 -14210.506,E2 -14210.506} C_VEL
LIN {X 0,Y 341.073,Z 246.001,A -85,B 0,C 180,E1 -14212.896,E2 -14212.896} C_VEL
LIN {X 0,Y 341.167,Z 245.987,A -85,B 0,C 180,E1 -14217.637,E2 -14217.637} C_VEL
LIN {X 0,Y 341.313,Z 245.97,A -85,B 0,C 180,E1 -14219.998,E2 -14219.998} C_VEL
LIN {X 0,Y 341.165,Z 245.99,A -85,B 0,C 180,E1 -14222.359,E2 -14222.359} C_VEL
LIN {X 0,Y 341.072,Z 246.003,A -85,B 0,C 180,E1 -14227.1,E2 -14227.1} C_VEL
LIN {X 0,Y 340.871,Z 246.028,A -85,B 0,C 180,E1 -14229.492,E2 -14229.492} C_VEL
LIN {X 0,Y 340.828,Z 246.353,A -85,B 0,C 180,E1 -14230.693,E2 -14230.693} C_VEL
LIN {X 0,Y 340.756,Z 248.978,A -85,B 0,C 180,E1 -14234.327,E2 -14234.327} C_VEL
LIN {X 0,Y 340.501,Z 252.024,A -85,B 0,C 180,E1 -14238.299,E2 -14238.299} C_VEL
LIN {X 0,Y 340.29,Z 254.843,A -85,B 0,C 180,E1 -14241.821,E2 -14241.821} C_VEL
LIN {X 0,Y 340.126,Z 257.789,A -85,B 0,C 180,E1 -14245.251,E2 -14245.251} C_VEL
LIN {X 0,Y 344.78,Z 271.877,A -85,B 0,C 180,E1 -14246.275,E2 -14246.275} C_VEL
LIN {X 0,Y 347.478,Z 282.558,A -85,B 0,C 180,E1 -14247.181,E2 -14247.181} C_VEL
LIN {X 0,Y 348.463,Z 287.366,A -85,B 0,C 180,E1 -14247.635,E2 -14247.635} C_VEL
LIN {X 0,Y 347.452,Z 297.814,A -85,B 0,C 180,E1 -14248.544,E2 -14248.544} C_VEL
LIN {X 0,Y 346.26,Z 308.563,A -85,B 0,C 180,E1 -14249.72,E2 -14249.72} C_VEL
LIN {X 0,Y 344.963,Z 319.064,A -85,B 0,C 180,E1 -14251.167,E2 -14251.167} C_VEL
LIN {X 0,Y 343.693,Z 328.386,A -85,B 0,C 180,E1 -14252.757,E2 -14252.757} C_VEL
LIN {X 0,Y 342.551,Z 336.506,A -85,B 0,C 180,E1 -14254.495,E2 -14254.495} C_VEL
LIN {X 0,Y 341.59,Z 342.985,A -85,B 0,C 180,E1 -14256.219,E2 -14256.219} C_VEL
LIN {X 0,Y 340.722,Z 348.911,A -85,B 0,C 180,E1 -14258.226,E2 -14258.226} C_VEL
LIN {X 0,Y 340.099,Z 353.16,A -85,B 0,C 180,E1 -14260.131,E2 -14260.131} C_VEL
LIN {X 0,Y 339.708,Z 355.954,A -85,B 0,C 180,E1 -14261.861,E2 -14261.861} C_VEL
LIN {X 0,Y 339.408,Z 357.805,A -85,B 0,C 180,E1 -14263.555,E2 -14263.555} C_VEL
LIN {X 0,Y 339.196,Z 358.823,A -85,B 0,C 180,E1 -14265.215,E2 -14265.215} C_VEL
LIN {X 0,Y 339.084,Z 359.078,A -85,B 0,C 180,E1 -14266.846,E2 -14266.846} C_VEL
LIN {X 0,Y 339.116,Z 358.564,A -85,B 0,C 180,E1 -14268.458,E2 -14268.458} C_VEL
LIN {X 0,Y 339.257,Z 357.321,A -85,B 0,C 180,E1 -14270.046,E2 -14270.046} C_VEL
LIN {X 0,Y 339.514,Z 355.003,A -85,B 0,C 180,E1 -14271.865,E2 -14271.865} C_VEL
LIN {X 0,Y 339.879,Z 351.527,A -85,B 0,C 180,E1 -14273.745,E2 -14273.745} C_VEL
LIN {X 0,Y 340.436,Z 346.743,A -85,B 0,C 180,E1 -14275.661,E2 -14275.661} C_VEL
LIN {X 0,Y 341.126,Z 340.343,A -85,B 0,C 180,E1 -14277.634,E2 -14277.634} C_VEL
LIN {X 0,Y 342.01,Z 333.044,A -85,B 0,C 180,E1 -14279.4,E2 -14279.4} C_VEL
LIN {X 0,Y 343.038,Z 324.174,A -85,B 0,C 180,E1 -14281.131,E2 -14281.131} C_VEL
LIN {X 0,Y 344.08,Z 314.567,A -85,B 0,C 180,E1 -14282.641,E2 -14282.641} C_VEL
LIN {X 0,Y 345.239,Z 303.277,A -85,B 0,C 180,E1 -14284.056,E2 -14284.056} C_VEL
LIN {X 0,Y 346.277,Z 291.63,A -85,B 0,C 180,E1 -14285.214,E2 -14285.214} C_VEL
LIN {X 0,Y 346.831,Z 284.884,A -85,B 0,C 180,E1 -14285.757,E2 -14285.757} C_VEL
LIN {X 0,Y 344.837,Z 274.723,A -85,B 0,C 180,E1 -14286.584,E2 -14286.584} C_VEL
LIN {X 0,Y 341.472,Z 261.644,A -85,B 0,C 180,E1 -14287.461,E2 -14287.461} C_VEL
LIN {X 0,Y 339.718,Z 255.143,A -85,B 0,C 180,E1 -14287.819,E2 -14287.819} C_VEL
LIN {X 0,Y 339.86,Z 251.17,A -85,B 0,C 180,E1 -14292.025,E2 -14292.025} C_VEL
LIN {X 0,Y 340.063,Z 247.291,A -85,B 0,C 180,E1 -14296.237,E2 -14296.237} C_VEL
LIN {X 0,Y 340.186,Z 246.114,A -85,B 0,C 180,E1 -14298.078,E2 -14298.078} C_VEL
LIN {X 0,Y 340.813,Z 246.031,A -85,B 0,C 180,E1 -14301.799,E2 -14301.799} C_VEL
LIN {X 0,Y 341.003,Z 246.006,A -85,B 0,C 180,E1 -14304.086,E2 -14304.086} C_VEL
LIN {X 0,Y 341.155,Z 245.989,A -85,B 0,C 180,E1 -14307.639,E2 -14307.639} C_VEL
LIN {X 0,Y 341.302,Z 245.969,A -85,B 0,C 180,E1 -14310.001,E2 -14310.001} C_VEL
LIN {X 0,Y 341.155,Z 245.986,A -85,B 0,C 180,E1 -14312.362,E2 -14312.362} C_VEL
LIN {X 0,Y 341.061,Z 246.004,A -85,B 0,C 180,E1 -14317.103,E2 -14317.103} C_VEL
LIN {X 0,Y 340.86,Z 246.025,A -85,B 0,C 180,E1 -14320.695,E2 -14320.695} C_VEL
LIN {X 0,Y 340.848,Z 246.025,A -85,B 0,C 180,E1 -14324.326,E2 -14324.326} C_VEL
LIN {X 0,Y 340.825,Z 246.029,A -85,B 0,C 180,E1 -14328.469,E2 -14328.469} C_VEL
LIN {X 0,Y 340.76,Z 246.035,A -85,B 0,C 180,E1 -14331.867,E2 -14331.867} C_VEL
LIN {X 0,Y 340.764,Z 246.035,A -85,B 0,C 180,E1 -14335.666,E2 -14335.666} C_VEL
LIN {X 0,Y 340.728,Z 246.041,A -85,B 0,C 180,E1 -14338.321,E2 -14338.321} C_VEL
LIN {X 0,Y 340.691,Z 246.047,A -85,B 0,C 180,E1 -14341.046,E2 -14341.046} C_VEL
LIN {X 0,Y 340.707,Z 246.043,A -85,B 0,C 180,E1 -14345.281,E2 -14345.281} C_VEL
LIN {X 0,Y 340.708,Z 246.046,A -85,B 0,C 180,E1 -14348.39,E2 -14348.39} C_VEL
LIN {X 0,Y 340.716,Z 246.041,A -85,B 0,C 180,E1 -14351.306,E2 -14351.306} C_VEL
LIN {X 0,Y 340.773,Z 246.04,A -85,B 0,C 180,E1 -14354.524,E2 -14354.524} C_VEL
LIN {X 0,Y 340.744,Z 246.039,A -85,B 0,C 180,E1 -14357.947,E2 -14357.947} C_VEL
LIN {X 0,Y 340.701,Z 246.042,A -85,B 0,C 180,E1 -14361.378,E2 -14361.378} C_VEL
LIN {X 0,Y 340.055,Z 246.129,A -85,B 0,C 180,E1 -14362.365,E2 -14362.365} C_VEL
LIN {X 0,Y 337.175,Z 246.484,A -85,B 0,C 180,E1 -14363.968,E2 -14363.968} C_VEL
LIN {X 0,Y 334.731,Z 246.786,A -85,B 0,C 180,E1 -14365.267,E2 -14365.267} C_VEL
LIN {X 0,Y 333.701,Z 246.92,A -85,B 0,C 180,E1 -14366.273,E2 -14366.273} C_VEL
LIN {X 0,Y 333.629,Z 246.924,A -85,B 0,C 180,E1 -14366.614,E2 -14366.614} C_VEL
LIN {X 0,Y 333.7,Z 246.916,A -85,B 0,C 180,E1 -14369.712,E2 -14369.712} C_VEL
LIN {X 0,Y 333.741,Z 246.914,A -85,B 0,C 180,E1 -14372.404,E2 -14372.404} C_VEL
LIN {X 0,Y 333.724,Z 246.912,A -85,B 0,C 180,E1 -14375.093,E2 -14375.093} C_VEL
LIN {X 0,Y 333.679,Z 246.917,A -85,B 0,C 180,E1 -14379.022,E2 -14379.022} C_VEL
LIN {X 0,Y 333.793,Z 246.905,A -85,B 0,C 180,E1 -14381.592,E2 -14381.592} C_VEL
LIN {X 0,Y 333.808,Z 246.903,A -85,B 0,C 180,E1 -14385.579,E2 -14385.579} C_VEL
LIN {X 0,Y 333.833,Z 246.898,A -85,B 0,C 180,E1 -14389.08,E2 -14389.08} C_VEL
LIN {X 0,Y 333.994,Z 246.878,A -85,B 0,C 180,E1 -14392.749,E2 -14392.749} C_VEL
LIN {X 0,Y 333.809,Z 246.902,A -85,B 0,C 180,E1 -14395.171,E2 -14395.171} C_VEL
LIN {X 0,Y 334.107,Z 246.868,A -85,B 0,C 180,E1 -14397.591,E2 -14397.591} C_VEL
LIN {X 0,Y 334.248,Z 246.85,A -85,B 0,C 180,E1 -14400.002,E2 -14400.002} C_VEL
LIN {X 0,Y 334.107,Z 246.865,A -85,B 0,C 180,E1 -14402.413,E2 -14402.413} C_VEL
LIN {X 0,Y 334,Z 246.88,A -85,B 0,C 180,E1 -14406.041,E2 -14406.041} C_VEL
LIN {X 0,Y 333.825,Z 246.904,A -85,B 0,C 180,E1 -14409.698,E2 -14409.698} C_VEL
LIN {X 0,Y 333.802,Z 246.907,A -85,B 0,C 180,E1 -14413.393,E2 -14413.393} C_VEL
LIN {X 0,Y 333.752,Z 246.911,A -85,B 0,C 180,E1 -14417.148,E2 -14417.148} C_VEL
LIN {X 0,Y 333.741,Z 246.913,A -85,B 0,C 180,E1 -14419.692,E2 -14419.692} C_VEL
LIN {X 0,Y 333.699,Z 246.915,A -85,B 0,C 180,E1 -14422.28,E2 -14422.28} C_VEL
LIN {X 0,Y 333.741,Z 246.91,A -85,B 0,C 180,E1 -14426.248,E2 -14426.248} C_VEL
LIN {X 0,Y 333.697,Z 246.918,A -85,B 0,C 180,E1 -14428.975,E2 -14428.975} C_VEL
LIN {X 0,Y 333.65,Z 246.922,A -85,B 0,C 180,E1 -14432.588,E2 -14432.588} C_VEL
LIN {X 0,Y 333.683,Z 246.917,A -85,B 0,C 180,E1 -14436.14,E2 -14436.14} C_VEL
LIN {X 0,Y 333.654,Z 246.926,A -85,B 0,C 180,E1 -14439.193,E2 -14439.193} C_VEL
LIN {X 0,Y 333.702,Z 247.036,A -85,B 0,C 180,E1 -14442.374,E2 -14442.374} C_VEL
LIN {X 0,Y 334.681,Z 252.434,A -85,B 0,C 180,E1 -14446.134,E2 -14446.134} C_VEL
LIN {X 0,Y 335.671,Z 257.631,A -85,B 0,C 180,E1 -14449.529,E2 -14449.529} C_VEL
LIN {X 0,Y 336.399,Z 262.756,A -85,B 0,C 180,E1 -14452.708,E2 -14452.708} C_VEL
LIN {X 0,Y 336.243,Z 266.045,A -85,B 0,C 180,E1 -14454.605,E2 -14454.605} C_VEL
LIN {X 0,Y 335.507,Z 271.63,A -85,B 0,C 180,E1 -14457.713,E2 -14457.713} C_VEL
LIN {X 0,Y 334.546,Z 279.468,A -85,B 0,C 180,E1 -14461.926,E2 -14461.926} C_VEL
LIN {X 0,Y 333.782,Z 286.793,A -85,B 0,C 180,E1 -14465.758,E2 -14465.758} C_VEL
LIN {X 0,Y 333.344,Z 292.068,A -85,B 0,C 180,E1 -14468.456,E2 -14468.456} C_VEL
LIN {X 0,Y 335.804,Z 306.528,A -85,B 0,C 180,E1 -14469.191,E2 -14469.191} C_VEL
LIN {X 0,Y 337.55,Z 320.086,A -85,B 0,C 180,E1 -14470.118,E2 -14470.118} C_VEL
LIN {X 0,Y 338.595,Z 331.2,A -85,B 0,C 180,E1 -14471.075,E2 -14471.075} C_VEL
LIN {X 0,Y 338.717,Z 334.509,A -85,B 0,C 180,E1 -14471.396,E2 -14471.396} C_VEL
LIN {X 0,Y 337.38,Z 345.734,A -85,B 0,C 180,E1 -14472.575,E2 -14472.575} C_VEL
LIN {X 0,Y 336.205,Z 355.929,A -85,B 0,C 180,E1 -14473.92,E2 -14473.92} C_VEL
LIN {X 0,Y 335.175,Z 365.121,A -85,B 0,C 180,E1 -14475.426,E2 -14475.426} C_VEL
LIN {X 0,Y 334.03,Z 374.079,A -85,B 0,C 180,E1 -14477.236,E2 -14477.236} C_VEL
LIN {X 0,Y 333.197,Z 381.298,A -85,B 0,C 180,E1 -14479.056,E2 -14479.056} C_VEL
LIN {X 0,Y 332.646,Z 387.057,A -85,B 0,C 180,E1 -14480.882,E2 -14480.882} C_VEL
LIN {X 0,Y 332.282,Z 391.583,A -85,B 0,C 180,E1 -14482.709,E2 -14482.709} C_VEL
LIN {X 0,Y 332.187,Z 393.967,A -85,B 0,C 180,E1 -14483.927,E2 -14483.927} C_VEL
LIN {X 0,Y 332.118,Z 395.912,A -85,B 0,C 180,E1 -14485.144,E2 -14485.144} C_VEL
LIN {X 0,Y 332.054,Z 397.427,A -85,B 0,C 180,E1 -14486.359,E2 -14486.359} C_VEL
LIN {X 0,Y 332.132,Z 399.138,A -85,B 0,C 180,E1 -14488.787,E2 -14488.787} C_VEL
LIN {X 0,Y 332.209,Z 399.397,A -85,B 0,C 180,E1 -14489.999,E2 -14489.999} C_VEL
LIN {X 0,Y 332.13,Z 399.245,A -85,B 0,C 180,E1 -14491.212,E2 -14491.212} C_VEL
LIN {X 0,Y 332.058,Z 397.662,A -85,B 0,C 180,E1 -14493.64,E2 -14493.64} C_VEL
LIN {X 0,Y 332.094,Z 396.27,A -85,B 0,C 180,E1 -14494.855,E2 -14494.855} C_VEL
LIN {X 0,Y 332.197,Z 393.352,A -85,B 0,C 180,E1 -14496.681,E2 -14496.681} C_VEL
LIN {X 0,Y 332.497,Z 389.405,A -85,B 0,C 180,E1 -14498.508,E2 -14498.508} C_VEL
LIN {X 0,Y 333.034,Z 384.334,A -85,B 0,C 180,E1 -14500.333,E2 -14500.333} C_VEL
LIN {X 0,Y 333.72,Z 377.989,A -85,B 0,C 180,E1 -14502.157,E2 -14502.157} C_VEL
LIN {X 0,Y 334.859,Z 370.134,A -85,B 0,C 180,E1 -14503.966,E2 -14503.966} C_VEL
LIN {X 0,Y 336.084,Z 360.367,A -85,B 0,C 180,E1 -14505.774,E2 -14505.774} C_VEL
LIN {X 0,Y 337.376,Z 350.345,A -85,B 0,C 180,E1 -14507.268,E2 -14507.268} C_VEL
LIN {X 0,Y 338.891,Z 339.102,A -85,B 0,C 180,E1 -14508.593,E2 -14508.593} C_VEL
LIN {X 0,Y 339.389,Z 333.184,A -85,B 0,C 180,E1 -14509.191,E2 -14509.191} C_VEL
LIN {X 0,Y 338.493,Z 320.846,A -85,B 0,C 180,E1 -14510.346,E2 -14510.346} C_VEL
LIN {X 0,Y 337.116,Z 308.476,A -85,B 0,C 180,E1 -14511.275,E2 -14511.275} C_VEL
LIN {X 0,Y 334.598,Z 295.781,A -85,B 0,C 180,E1 -14512.083,E2 -14512.083} C_VEL
LIN {X 0,Y 333.396,Z 290.348,A -85,B 0,C 180,E1 -14512.38,E2 -14512.38} C_VEL
LIN {X 0,Y 334.108,Z 283.01,A -85,B 0,C 180,E1 -14516.214,E2 -14516.214} C_VEL
LIN {X 0,Y 335.031,Z 275.643,A -85,B 0,C 180,E1 -14520.228,E2 -14520.228} C_VEL
LIN {X 0,Y 336.047,Z 268.436,A -85,B 0,C 180,E1 -14524.378,E2 -14524.378} C_VEL
LIN {X 0,Y 336.533,Z 264.917,A -85,B 0,C 180,E1 -14526.524,E2 -14526.524} C_VEL
LIN {X 0,Y 336.304,Z 261.434,A -85,B 0,C 180,E1 -14528.823,E2 -14528.823} C_VEL
LIN {X 0,Y 335.468,Z 256.954,A -85,B 0,C 180,E1 -14532.096,E2 -14532.096} C_VEL
LIN {X 0,Y 334.609,Z 251.971,A -85,B 0,C 180,E1 -14536.121,E2 -14536.121} C_VEL
LIN {X 0,Y 333.984,Z 248.594,A -85,B 0,C 180,E1 -14539.281,E2 -14539.281} C_VEL
LIN {X 0,Y 333.68,Z 246.922,A -85,B 0,C 180,E1 -14541.195,E2 -14541.195} C_VEL
LIN {X 0,Y 333.686,Z 246.92,A -85,B 0,C 180,E1 -14545.224,E2 -14545.224} C_VEL
LIN {X 0,Y 333.698,Z 246.92,A -85,B 0,C 180,E1 -14549.636,E2 -14549.636} C_VEL
LIN {X 0,Y 333.742,Z 246.914,A -85,B 0,C 180,E1 -14552.399,E2 -14552.399} C_VEL
LIN {X 0,Y 333.726,Z 246.916,A -85,B 0,C 180,E1 -14555.089,E2 -14555.089} C_VEL
LIN {X 0,Y 333.681,Z 246.921,A -85,B 0,C 180,E1 -14559.017,E2 -14559.017} C_VEL
LIN {X 0,Y 333.793,Z 246.905,A -85,B 0,C 180,E1 -14561.588,E2 -14561.588} C_VEL
LIN {X 0,Y 333.806,Z 246.907,A -85,B 0,C 180,E1 -14565.575,E2 -14565.575} C_VEL
LIN {X 0,Y 333.831,Z 246.899,A -85,B 0,C 180,E1 -14569.076,E2 -14569.076} C_VEL
LIN {X 0,Y 334.023,Z 246.88,A -85,B 0,C 180,E1 -14572.746,E2 -14572.746} C_VEL
LIN {X 0,Y 333.81,Z 246.905,A -85,B 0,C 180,E1 -14575.167,E2 -14575.167} C_VEL
LIN {X 0,Y 334.104,Z 246.866,A -85,B 0,C 180,E1 -14577.587,E2 -14577.587} C_VEL
LIN {X 0,Y 334.264,Z 246.848,A -85,B 0,C 180,E1 -14579.998,E2 -14579.998} C_VEL
LIN {X 0,Y 334.102,Z 246.869,A -85,B 0,C 180,E1 -14582.409,E2 -14582.409} C_VEL
LIN {X 0,Y 334.022,Z 246.881,A -85,B 0,C 180,E1 -14587.25,E2 -14587.25} C_VEL
LIN {X 0,Y 333.804,Z 246.909,A -85,B 0,C 180,E1 -14589.695,E2 -14589.695} C_VEL
LIN {X 0,Y 333.812,Z 248.559,A -85,B 0,C 180,E1 -14592.152,E2 -14592.152} C_VEL
LIN {X 0,Y 333.7,Z 250.338,A -85,B 0,C 180,E1 -14594.637,E2 -14594.637} C_VEL
LIN {X 0,Y 333.47,Z 253.237,A -85,B 0,C 180,E1 -14598.491,E2 -14598.491} C_VEL
LIN {X 0,Y 333.207,Z 256.252,A -85,B 0,C 180,E1 -14602.31,E2 -14602.31} C_VEL
LIN {X 0,Y 333.1,Z 258.194,A -85,B 0,C 180,E1 -14604.684,E2 -14604.684} C_VEL
LIN {X 0,Y 337.414,Z 270.976,A -85,B 0,C 180,E1 -14605.646,E2 -14605.646} C_VEL
LIN {X 0,Y 340.524,Z 282.65,A -85,B 0,C 180,E1 -14606.67,E2 -14606.67} C_VEL
LIN {X 0,Y 341.755,Z 289.542,A -85,B 0,C 180,E1 -14607.328,E2 -14607.328} C_VEL
LIN {X 0,Y 340.616,Z 300.34,A -85,B 0,C 180,E1 -14608.328,E2 -14608.328} C_VEL
LIN {X 0,Y 339.359,Z 310.956,A -85,B 0,C 180,E1 -14609.566,E2 -14609.566} C_VEL
LIN {X 0,Y 338.11,Z 320.596,A -85,B 0,C 180,E1 -14610.958,E2 -14610.958} C_VEL
LIN {X 0,Y 336.822,Z 329.274,A -85,B 0,C 180,E1 -14612.496,E2 -14612.496} C_VEL
LIN {X 0,Y 335.72,Z 336.692,A -85,B 0,C 180,E1 -14614.12,E2 -14614.12} C_VEL
LIN {X 0,Y 334.638,Z 343.658,A -85,B 0,C 180,E1 -14616.016,E2 -14616.016} C_VEL
LIN {X 0,Y 333.682,Z 349.84,A -85,B 0,C 180,E1 -14618.183,E2 -14618.183} C_VEL
LIN {X 0,Y 333.095,Z 353.517,A -85,B 0,C 180,E1 -14619.892,E2 -14619.892} C_VEL
LIN {X 0,Y 332.869,Z 355.215,A -85,B 0,C 180,E1 -14620.88,E2 -14620.88} C_VEL
LIN {X 0,Y 332.486,Z 357.419,A -85,B 0,C 180,E1 -14622.56,E2 -14622.56} C_VEL
LIN {X 0,Y 332.215,Z 358.848,A -85,B 0,C 180,E1 -14624.272,E2 -14624.272} C_VEL
LIN {X 0,Y 332.043,Z 359.486,A -85,B 0,C 180,E1 -14626.021,E2 -14626.021} C_VEL
LIN {X 0,Y 332.003,Z 359.286,A -85,B 0,C 180,E1 -14627.804,E2 -14627.804} C_VEL
LIN {X 0,Y 332.109,Z 358.186,A -85,B 0,C 180,E1 -14629.621,E2 -14629.621} C_VEL
LIN {X 0,Y 332.363,Z 356.105,A -85,B 0,C 180,E1 -14631.475,E2 -14631.475} C_VEL
LIN {X 0,Y 332.814,Z 352.133,A -85,B 0,C 180,E1 -14633.754,E2 -14633.754} C_VEL
LIN {X 0,Y 333.484,Z 346.408,A -85,B 0,C 180,E1 -14636.07,E2 -14636.07} C_VEL
LIN {X 0,Y 334.114,Z 340.735,A -85,B 0,C 180,E1 -14637.818,E2 -14637.818} C_VEL
LIN {X 0,Y 335.131,Z 332.69,A -85,B 0,C 180,E1 -14639.782,E2 -14639.782} C_VEL
LIN {X 0,Y 336.12,Z 324.371,A -85,B 0,C 180,E1 -14641.418,E2 -14641.418} C_VEL
LIN {X 0,Y 337.21,Z 314.931,A -85,B 0,C 180,E1 -14642.924,E2 -14642.924} C_VEL
LIN {X 0,Y 338.348,Z 304.18,A -85,B 0,C 180,E1 -14644.304,E2 -14644.304} C_VEL
LIN {X 0,Y 339.31,Z 293.932,A -85,B 0,C 180,E1 -14645.366,E2 -14645.366} C_VEL
LIN {X 0,Y 339.978,Z 285.681,A -85,B 0,C 180,E1 -14646.067,E2 -14646.067} C_VEL
LIN {X 0,Y 337.613,Z 274.124,A -85,B 0,C 180,E1 -14647.027,E2 -14647.027} C_VEL
LIN {X 0,Y 334.088,Z 260.868,A -85,B 0,C 180,E1 -14647.924,E2 -14647.924} C_VEL
LIN {X 0,Y 332.69,Z 255.522,A -85,B 0,C 180,E1 -14648.234,E2 -14648.234} C_VEL
LIN {X 0,Y 332.795,Z 252.146,A -85,B 0,C 180,E1 -14651.854,E2 -14651.854} C_VEL
LIN {X 0,Y 333.002,Z 248.261,A -85,B 0,C 180,E1 -14656.115,E2 -14656.115} C_VEL
LIN {X 0,Y 333.103,Z 246.997,A -85,B 0,C 180,E1 -14657.821,E2 -14657.821} C_VEL
LIN {X 0,Y 333.77,Z 246.909,A -85,B 0,C 180,E1 -14661.73,E2 -14661.73} C_VEL
LIN {X 0,Y 333.972,Z 246.882,A -85,B 0,C 180,E1 -14663.961,E2 -14663.961} C_VEL
LIN {X 0,Y 334.116,Z 246.866,A -85,B 0,C 180,E1 -14667.59,E2 -14667.59} C_VEL
LIN {X 0,Y 334.252,Z 246.846,A -85,B 0,C 180,E1 -14670.001,E2 -14670.001} C_VEL
LIN {X 0,Y 334.093,Z 246.866,A -85,B 0,C 180,E1 -14672.412,E2 -14672.412} C_VEL
LIN {X 0,Y 334.01,Z 246.881,A -85,B 0,C 180,E1 -14677.253,E2 -14677.253} C_VEL
LIN {X 0,Y 333.823,Z 246.904,A -85,B 0,C 180,E1 -14680.923,E2 -14680.923} C_VEL
LIN {X 0,Y 333.794,Z 246.905,A -85,B 0,C 180,E1 -14684.636,E2 -14684.636} C_VEL
LIN {X 0,Y 333.784,Z 246.907,A -85,B 0,C 180,E1 -14688.658,E2 -14688.658} C_VEL
LIN {X 0,Y 333.718,Z 246.913,A -85,B 0,C 180,E1 -14692.277,E2 -14692.277} C_VEL
LIN {X 0,Y 333.717,Z 246.916,A -85,B 0,C 180,E1 -14695.107,E2 -14695.107} C_VEL
LIN {X 0,Y 333.698,Z 246.919,A -85,B 0,C 180,E1 -14698.974,E2 -14698.974} C_VEL
LIN {X 0,Y 333.631,Z 246.928,A -85,B 0,C 180,E1 -14702.589,E2 -14702.589} C_VEL
LIN {X 0,Y 333.666,Z 246.92,A -85,B 0,C 180,E1 -14706.141,E2 -14706.141} C_VEL
LIN {X 0,Y 333.674,Z 246.919,A -85,B 0,C 180,E1 -14709.189,E2 -14709.189} C_VEL
LIN {X 0,Y 333.694,Z 246.921,A -85,B 0,C 180,E1 -14712.515,E2 -14712.515} C_VEL
LIN {X 0,Y 333.721,Z 246.914,A -85,B 0,C 180,E1 -14715.979,E2 -14715.979} C_VEL
LIN {X 0,Y 333.694,Z 246.916,A -85,B 0,C 180,E1 -14719.307,E2 -14719.307} C_VEL
LIN {X 0,Y 333.661,Z 246.92,A -85,B 0,C 180,E1 -14723.17,E2 -14723.17} C_VEL
LIN {X 0,Y 333.629,Z 246.924,A -85,B 0,C 180,E1 -14726.614,E2 -14726.614} C_VEL
LIN {X 0,Y 333.002,Z 247.009,A -85,B 0,C 180,E1 -14727.622,E2 -14727.622} C_VEL
LIN {X 0,Y 330.198,Z 247.365,A -85,B 0,C 180,E1 -14729.263,E2 -14729.263} C_VEL
LIN {X 0,Y 327.793,Z 247.661,A -85,B 0,C 180,E1 -14730.592,E2 -14730.592} C_VEL
LIN {X 0,Y 326.747,Z 247.786,A -85,B 0,C 180,E1 -14731.62,E2 -14731.62} C_VEL
LIN {X 0,Y 326.655,Z 247.794,A -85,B 0,C 180,E1 -14731.969,E2 -14731.969} C_VEL
LIN {X 0,Y 326.685,Z 247.79,A -85,B 0,C 180,E1 -14734.63,E2 -14734.63} C_VEL
LIN {X 0,Y 326.644,Z 247.795,A -85,B 0,C 180,E1 -14738.548,E2 -14738.548} C_VEL
LIN {X 0,Y 326.743,Z 247.781,A -85,B 0,C 180,E1 -14741.18,E2 -14741.18} C_VEL
LIN {X 0,Y 326.763,Z 247.78,A -85,B 0,C 180,E1 -14745.435,E2 -14745.435} C_VEL
LIN {X 0,Y 326.769,Z 247.778,A -85,B 0,C 180,E1 -14748.841,E2 -14748.841} C_VEL
LIN {X 0,Y 326.944,Z 247.757,A -85,B 0,C 180,E1 -14752.592,E2 -14752.592} C_VEL
LIN {X 0,Y 326.984,Z 247.757,A -85,B 0,C 180,E1 -14753.833,E2 -14753.833} C_VEL
LIN {X 0,Y 327.048,Z 247.746,A -85,B 0,C 180,E1 -14757.539,E2 -14757.539} C_VEL
LIN {X 0,Y 327.2,Z 247.728,A -85,B 0,C 180,E1 -14760.002,E2 -14760.002} C_VEL
LIN {X 0,Y 327.048,Z 247.744,A -85,B 0,C 180,E1 -14762.465,E2 -14762.465} C_VEL
LIN {X 0,Y 326.954,Z 247.756,A -85,B 0,C 180,E1 -14766.172,E2 -14766.172} C_VEL
LIN {X 0,Y 326.788,Z 247.779,A -85,B 0,C 180,E1 -14769.909,E2 -14769.909} C_VEL
LIN {X 0,Y 326.764,Z 247.783,A -85,B 0,C 180,E1 -14773.687,E2 -14773.687} C_VEL
LIN {X 0,Y 326.705,Z 247.791,A -85,B 0,C 180,E1 -14777.529,E2 -14777.529} C_VEL
LIN {X 0,Y 326.667,Z 247.791,A -85,B 0,C 180,E1 -14780.137,E2 -14780.137} C_VEL
LIN {X 0,Y 326.658,Z 247.792,A -85,B 0,C 180,E1 -14784.13,E2 -14784.13} C_VEL
LIN {X 0,Y 326.689,Z 247.79,A -85,B 0,C 180,E1 -14786.859,E2 -14786.859} C_VEL
LIN {X 0,Y 326.641,Z 247.795,A -85,B 0,C 180,E1 -14790.611,E2 -14790.611} C_VEL
LIN {X 0,Y 326.614,Z 247.798,A -85,B 0,C 180,E1 -14794.02,E2 -14794.02} C_VEL
LIN {X 0,Y 326.634,Z 247.8,A -85,B 0,C 180,E1 -14797.239,E2 -14797.239} C_VEL
LIN {X 0,Y 326.607,Z 247.803,A -85,B 0,C 180,E1 -14801.137,E2 -14801.137} C_VEL
LIN {X 0,Y 326.683,Z 248.002,A -85,B 0,C 180,E1 -14802.038,E2 -14802.038} C_VEL
LIN {X 0,Y 327.653,Z 253.406,A -85,B 0,C 180,E1 -14805.886,E2 -14805.886} C_VEL
LIN {X 0,Y 328.612,Z 258.509,A -85,B 0,C 180,E1 -14809.322,E2 -14809.322} C_VEL
LIN {X 0,Y 329.288,Z 262.972,A -85,B 0,C 180,E1 -14812.159,E2 -14812.159} C_VEL
LIN {X 0,Y 329.286,Z 266.393,A -85,B 0,C 180,E1 -14814.2,E2 -14814.2} C_VEL
LIN {X 0,Y 328.464,Z 272.462,A -85,B 0,C 180,E1 -14817.661,E2 -14817.661} C_VEL
LIN {X 0,Y 327.545,Z 279.641,A -85,B 0,C 180,E1 -14821.611,E2 -14821.611} C_VEL
LIN {X 0,Y 326.817,Z 286.316,A -85,B 0,C 180,E1 -14825.207,E2 -14825.207} C_VEL
LIN {X 0,Y 326.335,Z 291.709,A -85,B 0,C 180,E1 -14828.047,E2 -14828.047} C_VEL
LIN {X 0,Y 328.654,Z 305.485,A -85,B 0,C 180,E1 -14828.74,E2 -14828.74} C_VEL
LIN {X 0,Y 330.465,Z 318.532,A -85,B 0,C 180,E1 -14829.64,E2 -14829.64} C_VEL
LIN {X 0,Y 331.523,Z 330.236,A -85,B 0,C 180,E1 -14830.656,E2 -14830.656} C_VEL
LIN {X 0,Y 331.789,Z 335.203,A -85,B 0,C 180,E1 -14831.153,E2 -14831.153} C_VEL
LIN {X 0,Y 330.418,Z 346.223,A -85,B 0,C 180,E1 -14832.356,E2 -14832.356} C_VEL
LIN {X 0,Y 329.329,Z 355.206,A -85,B 0,C 180,E1 -14833.574,E2 -14833.574} C_VEL
LIN {X 0,Y 328.282,Z 364.465,A -85,B 0,C 180,E1 -14835.113,E2 -14835.113} C_VEL
LIN {X 0,Y 327.072,Z 373.461,A -85,B 0,C 180,E1 -14836.96,E2 -14836.96} C_VEL
LIN {X 0,Y 326.161,Z 380.715,A -85,B 0,C 180,E1 -14838.817,E2 -14838.817} C_VEL
LIN {X 0,Y 325.609,Z 386.517,A -85,B 0,C 180,E1 -14840.683,E2 -14840.683} C_VEL
LIN {X 0,Y 325.211,Z 391.071,A -85,B 0,C 180,E1 -14842.549,E2 -14842.549} C_VEL
LIN {X 0,Y 325.109,Z 393.729,A -85,B 0,C 180,E1 -14843.945,E2 -14843.945} C_VEL
LIN {X 0,Y 324.983,Z 396.958,A -85,B 0,C 180,E1 -14846.28,E2 -14846.28} C_VEL
LIN {X 0,Y 324.952,Z 398.029,A -85,B 0,C 180,E1 -14847.52,E2 -14847.52} C_VEL
LIN {X 0,Y 325.039,Z 398.695,A -85,B 0,C 180,E1 -14848.76,E2 -14848.76} C_VEL
LIN {X 0,Y 325.135,Z 398.965,A -85,B 0,C 180,E1 -14849.999,E2 -14849.999} C_VEL
LIN {X 0,Y 325.036,Z 398.827,A -85,B 0,C 180,E1 -14851.238,E2 -14851.238} C_VEL
LIN {X 0,Y 324.951,Z 398.249,A -85,B 0,C 180,E1 -14852.478,E2 -14852.478} C_VEL
LIN {X 0,Y 324.985,Z 397.268,A -85,B 0,C 180,E1 -14853.719,E2 -14853.719} C_VEL
LIN {X 0,Y 325.084,Z 394.378,A -85,B 0,C 180,E1 -14856.015,E2 -14856.015} C_VEL
LIN {X 0,Y 325.304,Z 390.515,A -85,B 0,C 180,E1 -14858.072,E2 -14858.072} C_VEL
LIN {X 0,Y 325.806,Z 385.868,A -85,B 0,C 180,E1 -14859.936,E2 -14859.936} C_VEL
LIN {X 0,Y 326.582,Z 378.869,A -85,B 0,C 180,E1 -14862.111,E2 -14862.111} C_VEL
LIN {X 0,Y 327.746,Z 371.34,A -85,B 0,C 180,E1 -14863.959,E2 -14863.959} C_VEL
LIN {X 0,Y 328.901,Z 362.995,A -85,B 0,C 180,E1 -14865.629,E2 -14865.629} C_VEL
LIN {X 0,Y 330.111,Z 353.475,A -85,B 0,C 180,E1 -14867.18,E2 -14867.18} C_VEL
LIN {X 0,Y 331.773,Z 341.832,A -85,B 0,C 180,E1 -14868.686,E2 -14868.686} C_VEL
LIN {X 0,Y 332.626,Z 334.836,A -85,B 0,C 180,E1 -14869.437,E2 -14869.437} C_VEL
LIN {X 0,Y 331.782,Z 321.444,A -85,B 0,C 180,E1 -14870.751,E2 -14870.751} C_VEL
LIN {X 0,Y 330.497,Z 309.674,A -85,B 0,C 180,E1 -14871.699,E2 -14871.699} C_VEL
LIN {X 0,Y 328.193,Z 297.445,A -85,B 0,C 180,E1 -14872.53,E2 -14872.53} C_VEL
LIN {X 0,Y 326.413,Z 289.885,A -85,B 0,C 180,E1 -14872.969,E2 -14872.969} C_VEL
LIN {X 0,Y 327.027,Z 283.972,A -85,B 0,C 180,E1 -14876.139,E2 -14876.139} C_VEL
LIN {X 0,Y 327.982,Z 276.64,A -85,B 0,C 180,E1 -14880.235,E2 -14880.235} C_VEL
LIN {X 0,Y 328.878,Z 270.656,A -85,B 0,C 180,E1 -14883.752,E2 -14883.752} C_VEL
LIN {X 0,Y 329.557,Z 265.948,A -85,B 0,C 180,E1 -14886.663,E2 -14886.663} C_VEL
LIN {X 0,Y 329.316,Z 262.565,A -85,B 0,C 180,E1 -14888.977,E2 -14888.977} C_VEL
LIN {X 0,Y 328.272,Z 256.911,A -85,B 0,C 180,E1 -14893.241,E2 -14893.241} C_VEL
LIN {X 0,Y 327.54,Z 252.75,A -85,B 0,C 180,E1 -14896.846,E2 -14896.846} C_VEL
LIN {X 0,Y 326.793,Z 248.847,A -85,B 0,C 180,E1 -14900.732,E2 -14900.732} C_VEL
LIN {X 0,Y 326.636,Z 247.8,A -85,B 0,C 180,E1 -14902.134,E2 -14902.134} C_VEL
LIN {X 0,Y 326.608,Z 247.805,A -85,B 0,C 180,E1 -14905.979,E2 -14905.979} C_VEL
LIN {X 0,Y 326.661,Z 247.795,A -85,B 0,C 180,E1 -14910.339,E2 -14910.339} C_VEL
LIN {X 0,Y 326.69,Z 247.792,A -85,B 0,C 180,E1 -14914.514,E2 -14914.514} C_VEL
LIN {X 0,Y 326.646,Z 247.798,A -85,B 0,C 180,E1 -14918.543,E2 -14918.543} C_VEL
LIN {X 0,Y 326.743,Z 247.785,A -85,B 0,C 180,E1 -14921.176,E2 -14921.176} C_VEL
LIN {X 0,Y 326.761,Z 247.784,A -85,B 0,C 180,E1 -14925.431,E2 -14925.431} C_VEL
LIN {X 0,Y 326.767,Z 247.78,A -85,B 0,C 180,E1 -14928.837,E2 -14928.837} C_VEL
LIN {X 0,Y 326.977,Z 247.757,A -85,B 0,C 180,E1 -14932.588,E2 -14932.588} C_VEL
LIN {X 0,Y 326.777,Z 247.781,A -85,B 0,C 180,E1 -14935.063,E2 -14935.063} C_VEL
LIN {X 0,Y 327.045,Z 247.746,A -85,B 0,C 180,E1 -14937.535,E2 -14937.535} C_VEL
LIN {X 0,Y 327.214,Z 247.726,A -85,B 0,C 180,E1 -14939.998,E2 -14939.998} C_VEL
LIN {X 0,Y 327.043,Z 247.748,A -85,B 0,C 180,E1 -14942.461,E2 -14942.461} C_VEL
LIN {X 0,Y 326.966,Z 247.758,A -85,B 0,C 180,E1 -14946.674,E2 -14946.674} C_VEL
LIN {X 0,Y 326.906,Z 247.766,A -85,B 0,C 180,E1 -14948.653,E2 -14948.653} C_VEL
LIN {X 0,Y 326.822,Z 249.062,A -85,B 0,C 180,E1 -14951.157,E2 -14951.157} C_VEL
LIN {X 0,Y 326.672,Z 251.7,A -85,B 0,C 180,E1 -14954.959,E2 -14954.959} C_VEL
LIN {X 0,Y 326.411,Z 254.572,A -85,B 0,C 180,E1 -14958.84,E2 -14958.84} C_VEL
LIN {X 0,Y 326.155,Z 257.661,A -85,B 0,C 180,E1 -14962.819,E2 -14962.819} C_VEL
LIN {X 0,Y 326.116,Z 258.675,A -85,B 0,C 180,E1 -14964.084,E2 -14964.084} C_VEL
LIN {X 0,Y 330.82,Z 272.509,A -85,B 0,C 180,E1 -14965.188,E2 -14965.188} C_VEL
LIN {X 0,Y 333.854,Z 283.869,A -85,B 0,C 180,E1 -14966.234,E2 -14966.234} C_VEL
LIN {X 0,Y 335.084,Z 289.863,A -85,B 0,C 180,E1 -14966.843,E2 -14966.843} C_VEL
LIN {X 0,Y 334,Z 300.937,A -85,B 0,C 180,E1 -14967.903,E2 -14967.903} C_VEL
LIN {X 0,Y 332.633,Z 312.083,A -85,B 0,C 180,E1 -14969.239,E2 -14969.239} C_VEL
LIN {X 0,Y 331.355,Z 321.24,A -85,B 0,C 180,E1 -14970.597,E2 -14970.597} C_VEL
LIN {X 0,Y 330.009,Z 329.882,A -85,B 0,C 180,E1 -14972.165,E2 -14972.165} C_VEL
LIN {X 0,Y 328.91,Z 336.974,A -85,B 0,C 180,E1 -14973.746,E2 -14973.746} C_VEL
LIN {X 0,Y 327.707,Z 344.241,A -85,B 0,C 180,E1 -14975.765,E2 -14975.765} C_VEL
LIN {X 0,Y 326.714,Z 350.236,A -85,B 0,C 180,E1 -14977.917,E2 -14977.917} C_VEL
LIN {X 0,Y 326.091,Z 353.944,A -85,B 0,C 180,E1 -14979.679,E2 -14979.679} C_VEL
LIN {X 0,Y 325.519,Z 357.41,A -85,B 0,C 180,E1 -14982.009,E2 -14982.009} C_VEL
LIN {X 0,Y 325.11,Z 359.483,A -85,B 0,C 180,E1 -14984.492,E2 -14984.492} C_VEL
LIN {X 0,Y 324.958,Z 359.943,A -85,B 0,C 180,E1 -14986.207,E2 -14986.207} C_VEL
LIN {X 0,Y 324.915,Z 359.668,A -85,B 0,C 180,E1 -14987.893,E2 -14987.893} C_VEL
LIN {X 0,Y 325.025,Z 358.675,A -85,B 0,C 180,E1 -14989.558,E2 -14989.558} C_VEL
LIN {X 0,Y 325.374,Z 355.813,A -85,B 0,C 180,E1 -14992.006,E2 -14992.006} C_VEL
LIN {X 0,Y 325.892,Z 351.423,A -85,B 0,C 180,E1 -14994.391,E2 -14994.391} C_VEL
LIN {X 0,Y 326.55,Z 345.866,A -85,B 0,C 180,E1 -14996.535,E2 -14996.535} C_VEL
LIN {X 0,Y 327.436,Z 338.798,A -85,B 0,C 180,E1 -14998.635,E2 -14998.635} C_VEL
LIN {X 0,Y 328.456,Z 330.699,A -85,B 0,C 180,E1 -15000.52,E2 -15000.52} C_VEL
LIN {X 0,Y 329.679,Z 320.788,A -85,B 0,C 180,E1 -15002.36,E2 -15002.36} C_VEL
LIN {X 0,Y 330.809,Z 310.784,A -85,B 0,C 180,E1 -15003.844,E2 -15003.844} C_VEL
LIN {X 0,Y 332.088,Z 298.905,A -85,B 0,C 180,E1 -15005.243,E2 -15005.243} C_VEL
LIN {X 0,Y 333.118,Z 286.659,A -85,B 0,C 180,E1 -15006.369,E2 -15006.369} C_VEL
LIN {X 0,Y 330.72,Z 275.076,A -85,B 0,C 180,E1 -15007.367,E2 -15007.367} C_VEL
LIN {X 0,Y 327.208,Z 261.744,A -85,B 0,C 180,E1 -15008.305,E2 -15008.305} C_VEL
LIN {X 0,Y 325.622,Z 255.93,A -85,B 0,C 180,E1 -15008.641,E2 -15008.641} C_VEL
LIN {X 0,Y 325.769,Z 252.447,A -85,B 0,C 180,E1 -15012.421,E2 -15012.421} C_VEL
LIN {X 0,Y 325.963,Z 248.989,A -85,B 0,C 180,E1 -15016.281,E2 -15016.281} C_VEL
LIN {X 0,Y 326.032,Z 247.881,A -85,B 0,C 180,E1 -15017.552,E2 -15017.552} C_VEL
LIN {X 0,Y 326.723,Z 247.787,A -85,B 0,C 180,E1 -15021.664,E2 -15021.664} C_VEL
LIN {X 0,Y 326.92,Z 247.761,A -85,B 0,C 180,E1 -15023.83,E2 -15023.83} C_VEL
LIN {X 0,Y 327.053,Z 247.746,A -85,B 0,C 180,E1 -15027.537,E2 -15027.537} C_VEL
LIN {X 0,Y 327.203,Z 247.725,A -85,B 0,C 180,E1 -15030.001,E2 -15030.001} C_VEL
LIN {X 0,Y 327.033,Z 247.745,A -85,B 0,C 180,E1 -15032.464,E2 -15032.464} C_VEL
LIN {X 0,Y 326.982,Z 247.751,A -85,B 0,C 180,E1 -15036.17,E2 -15036.17} C_VEL
LIN {X 0,Y 326.9,Z 247.763,A -85,B 0,C 180,E1 -15038.656,E2 -15038.656} C_VEL
LIN {X 0,Y 326.724,Z 247.784,A -85,B 0,C 180,E1 -15042.422,E2 -15042.422} C_VEL
LIN {X 0,Y 326.74,Z 247.787,A -85,B 0,C 180,E1 -15044.959,E2 -15044.959} C_VEL
LIN {X 0,Y 326.75,Z 247.785,A -85,B 0,C 180,E1 -15048.856,E2 -15048.856} C_VEL
LIN {X 0,Y 326.673,Z 247.795,A -85,B 0,C 180,E1 -15052.784,E2 -15052.784} C_VEL
LIN {X 0,Y 326.672,Z 247.796,A -85,B 0,C 180,E1 -15056.859,E2 -15056.859} C_VEL
LIN {X 0,Y 326.627,Z 247.8,A -85,B 0,C 180,E1 -15060.613,E2 -15060.613} C_VEL
LIN {X 0,Y 326.596,Z 247.8,A -85,B 0,C 180,E1 -15064.021,E2 -15064.021} C_VEL
LIN {X 0,Y 326.619,Z 247.798,A -85,B 0,C 180,E1 -15067.241,E2 -15067.241} C_VEL
LIN {X 0,Y 326.625,Z 247.798,A -85,B 0,C 180,E1 -15070.205,E2 -15070.205} C_VEL
LIN {X 0,Y 326.649,Z 247.793,A -85,B 0,C 180,E1 -15073.512,E2 -15073.512} C_VEL
LIN {X 0,Y 326.642,Z 247.795,A -85,B 0,C 180,E1 -15077.016,E2 -15077.016} C_VEL
LIN {X 0,Y 326.638,Z 247.797,A -85,B 0,C 180,E1 -15080.768,E2 -15080.768} C_VEL
LIN {X 0,Y 326.608,Z 247.803,A -85,B 0,C 180,E1 -15084.483,E2 -15084.483} C_VEL
LIN {X 0,Y 326.61,Z 247.798,A -85,B 0,C 180,E1 -15087.459,E2 -15087.459} C_VEL
LIN {X 0,Y 326.657,Z 247.797,A -85,B 0,C 180,E1 -15090.343,E2 -15090.343} C_VEL
LIN {X 0,Y 326.655,Z 247.794,A -85,B 0,C 180,E1 -15091.969,E2 -15091.969} C_VEL
LIN {X 0,Y 325.955,Z 247.88,A -85,B 0,C 180,E1 -15092.998,E2 -15092.998} C_VEL
LIN {X 0,Y 323.053,Z 248.242,A -85,B 0,C 180,E1 -15094.672,E2 -15094.672} C_VEL
LIN {X 0,Y 320.643,Z 248.546,A -85,B 0,C 180,E1 -15096.029,E2 -15096.029} C_VEL
LIN {X 0,Y 319.659,Z 248.664,A -85,B 0,C 180,E1 -15097.08,E2 -15097.08} C_VEL
LIN {X 0,Y 319.605,Z 248.671,A -85,B 0,C 180,E1 -15097.436,E2 -15097.436} C_VEL
LIN {X 0,Y 319.688,Z 248.66,A -85,B 0,C 180,E1 -15100.965,E2 -15100.965} C_VEL
LIN {X 0,Y 319.73,Z 248.655,A -85,B 0,C 180,E1 -15105.278,E2 -15105.278} C_VEL
LIN {X 0,Y 319.752,Z 248.657,A -85,B 0,C 180,E1 -15109.875,E2 -15109.875} C_VEL
LIN {X 0,Y 319.938,Z 248.633,A -85,B 0,C 180,E1 -15113.696,E2 -15113.696} C_VEL
LIN {X 0,Y 319.991,Z 248.624,A -85,B 0,C 180,E1 -15117.485,E2 -15117.485} C_VEL
LIN {X 0,Y 320.152,Z 248.606,A -85,B 0,C 180,E1 -15120.002,E2 -15120.002} C_VEL
LIN {X 0,Y 319.991,Z 248.623,A -85,B 0,C 180,E1 -15122.52,E2 -15122.52} C_VEL
LIN {X 0,Y 319.91,Z 248.632,A -85,B 0,C 180,E1 -15126.308,E2 -15126.308} C_VEL
LIN {X 0,Y 319.74,Z 248.655,A -85,B 0,C 180,E1 -15130.13,E2 -15130.13} C_VEL
LIN {X 0,Y 319.738,Z 248.655,A -85,B 0,C 180,E1 -15133.994,E2 -15133.994} C_VEL
LIN {X 0,Y 319.664,Z 248.665,A -85,B 0,C 180,E1 -15137.928,E2 -15137.928} C_VEL
LIN {X 0,Y 319.619,Z 248.669,A -85,B 0,C 180,E1 -15140.601,E2 -15140.601} C_VEL
LIN {X 0,Y 319.576,Z 248.679,A -85,B 0,C 180,E1 -15143.321,E2 -15143.321} C_VEL
LIN {X 0,Y 319.625,Z 248.668,A -85,B 0,C 180,E1 -15146.091,E2 -15146.091} C_VEL
LIN {X 0,Y 319.587,Z 248.675,A -85,B 0,C 180,E1 -15148.936,E2 -15148.936} C_VEL
LIN {X 0,Y 319.538,Z 248.68,A -85,B 0,C 180,E1 -15151.863,E2 -15151.863} C_VEL
LIN {X 0,Y 319.587,Z 248.675,A -85,B 0,C 180,E1 -15155.544,E2 -15155.544} C_VEL
LIN {X 0,Y 319.564,Z 248.681,A -85,B 0,C 180,E1 -15158.011,E2 -15158.011} C_VEL
LIN {X 0,Y 319.627,Z 248.854,A -85,B 0,C 180,E1 -15161.617,E2 -15161.617} C_VEL
LIN {X 0,Y 320.565,Z 254.081,A -85,B 0,C 180,E1 -15165.447,E2 -15165.447} C_VEL
LIN {X 0,Y 321.554,Z 259.276,A -85,B 0,C 180,E1 -15169.027,E2 -15169.027} C_VEL
LIN {X 0,Y 322.306,Z 264.432,A -85,B 0,C 180,E1 -15172.37,E2 -15172.37} C_VEL
LIN {X 0,Y 322.129,Z 268.238,A -85,B 0,C 180,E1 -15174.678,E2 -15174.678} C_VEL
LIN {X 0,Y 321.432,Z 273.263,A -85,B 0,C 180,E1 -15177.609,E2 -15177.609} C_VEL
LIN {X 0,Y 320.553,Z 279.782,A -85,B 0,C 180,E1 -15181.283,E2 -15181.283} C_VEL
LIN {X 0,Y 319.717,Z 287.101,A -85,B 0,C 180,E1 -15185.313,E2 -15185.313} C_VEL
LIN {X 0,Y 319.291,Z 291.33,A -85,B 0,C 180,E1 -15187.592,E2 -15187.592} C_VEL
LIN {X 0,Y 321.728,Z 305.707,A -85,B 0,C 180,E1 -15188.36,E2 -15188.36} C_VEL
LIN {X 0,Y 323.59,Z 319.372,A -85,B 0,C 180,E1 -15189.346,E2 -15189.346} C_VEL
LIN {X 0,Y 324.62,Z 330.948,A -85,B 0,C 180,E1 -15190.392,E2 -15190.392} C_VEL
LIN {X 0,Y 324.878,Z 335.821,A -85,B 0,C 180,E1 -15190.901,E2 -15190.901} C_VEL
LIN {X 0,Y 323.459,Z 346.604,A -85,B 0,C 180,E1 -15192.127,E2 -15192.127} C_VEL
LIN {X 0,Y 322.222,Z 356.436,A -85,B 0,C 180,E1 -15193.528,E2 -15193.528} C_VEL
LIN {X 0,Y 321.142,Z 365.414,A -85,B 0,C 180,E1 -15195.099,E2 -15195.099} C_VEL
LIN {X 0,Y 319.932,Z 374.181,A -85,B 0,C 180,E1 -15196.987,E2 -15196.987} C_VEL
LIN {X 0,Y 319.047,Z 381.181,A -85,B 0,C 180,E1 -15198.886,E2 -15198.886} C_VEL
LIN {X 0,Y 318.393,Z 387.602,A -85,B 0,C 180,E1 -15201.111,E2 -15201.111} C_VEL
LIN {X 0,Y 318.078,Z 391.81,A -85,B 0,C 180,E1 -15203.019,E2 -15203.019} C_VEL
LIN {X 0,Y 317.953,Z 394.938,A -85,B 0,C 180,E1 -15204.927,E2 -15204.927} C_VEL
LIN {X 0,Y 317.915,Z 396.485,A -85,B 0,C 180,E1 -15206.197,E2 -15206.197} C_VEL
LIN {X 0,Y 317.868,Z 397.576,A -85,B 0,C 180,E1 -15207.465,E2 -15207.465} C_VEL
LIN {X 0,Y 317.946,Z 398.252,A -85,B 0,C 180,E1 -15208.733,E2 -15208.733} C_VEL
LIN {X 0,Y 318.046,Z 398.533,A -85,B 0,C 180,E1 -15209.999,E2 -15209.999} C_VEL
LIN {X 0,Y 317.942,Z 398.406,A -85,B 0,C 180,E1 -15211.266,E2 -15211.266} C_VEL
LIN {X 0,Y 317.867,Z 397.85,A -85,B 0,C 180,E1 -15212.534,E2 -15212.534} C_VEL
LIN {X 0,Y 317.914,Z 396.882,A -85,B 0,C 180,E1 -15213.802,E2 -15213.802} C_VEL
LIN {X 0,Y 318.025,Z 393.732,A -85,B 0,C 180,E1 -15216.343,E2 -15216.343} C_VEL
LIN {X 0,Y 318.245,Z 390.186,A -85,B 0,C 180,E1 -15218.252,E2 -15218.252} C_VEL
LIN {X 0,Y 318.762,Z 385.568,A -85,B 0,C 180,E1 -15220.158,E2 -15220.158} C_VEL
LIN {X 0,Y 319.608,Z 378.619,A -85,B 0,C 180,E1 -15222.379,E2 -15222.379} C_VEL
LIN {X 0,Y 320.831,Z 371.127,A -85,B 0,C 180,E1 -15224.266,E2 -15224.266} C_VEL
LIN {X 0,Y 322.102,Z 362.331,A -85,B 0,C 180,E1 -15226.065,E2 -15226.065} C_VEL
LIN {X 0,Y 323.486,Z 352.338,A -85,B 0,C 180,E1 -15227.707,E2 -15227.707} C_VEL
LIN {X 0,Y 325.065,Z 341.879,A -85,B 0,C 180,E1 -15229.086,E2 -15229.086} C_VEL
LIN {X 0,Y 325.825,Z 335.022,A -85,B 0,C 180,E1 -15229.859,E2 -15229.859} C_VEL
LIN {X 0,Y 325.122,Z 322.211,A -85,B 0,C 180,E1 -15231.167,E2 -15231.167} C_VEL
LIN {X 0,Y 323.799,Z 309.906,A -85,B 0,C 180,E1 -15232.204,E2 -15232.204} C_VEL
LIN {X 0,Y 321.359,Z 297.334,A -85,B 0,C 180,E1 -15233.107,E2 -15233.107} C_VEL
LIN {X 0,Y 319.467,Z 289.358,A -85,B 0,C 180,E1 -15233.606,E2 -15233.606} C_VEL
LIN {X 0,Y 320.236,Z 282.485,A -85,B 0,C 180,E1 -15237.442,E2 -15237.442} C_VEL
LIN {X 0,Y 321.08,Z 276.626,A -85,B 0,C 180,E1 -15240.838,E2 -15240.838} C_VEL
LIN {X 0,Y 322.059,Z 270.496,A -85,B 0,C 180,E1 -15244.566,E2 -15244.566} C_VEL
LIN {X 0,Y 322.502,Z 267.822,A -85,B 0,C 180,E1 -15246.261,E2 -15246.261} C_VEL
LIN {X 0,Y 322.436,Z 264.838,A -85,B 0,C 180,E1 -15248.307,E2 -15248.307} C_VEL
LIN {X 0,Y 321.863,Z 261.329,A -85,B 0,C 180,E1 -15250.923,E2 -15250.923} C_VEL
LIN {X 0,Y 321.085,Z 256.973,A -85,B 0,C 180,E1 -15254.46,E2 -15254.46} C_VEL
LIN {X 0,Y 320.363,Z 252.85,A -85,B 0,C 180,E1 -15258.233,E2 -15258.233} C_VEL
LIN {X 0,Y 319.662,Z 249.082,A -85,B 0,C 180,E1 -15262.323,E2 -15262.323} C_VEL
LIN {X 0,Y 319.601,Z 248.676,A -85,B 0,C 180,E1 -15262.948,E2 -15262.948} C_VEL
LIN {X 0,Y 319.578,Z 248.677,A -85,B 0,C 180,E1 -15266.685,E2 -15266.685} C_VEL
LIN {X 0,Y 319.592,Z 248.677,A -85,B 0,C 180,E1 -15269.615,E2 -15269.615} C_VEL
LIN {X 0,Y 319.608,Z 248.674,A -85,B 0,C 180,E1 -15272.496,E2 -15272.496} C_VEL
LIN {X 0,Y 319.605,Z 248.676,A -85,B 0,C 180,E1 -15275.302,E2 -15275.302} C_VEL
LIN {X 0,Y 319.596,Z 248.673,A -85,B 0,C 180,E1 -15278.046,E2 -15278.046} C_VEL
LIN {X 0,Y 319.688,Z 248.664,A -85,B 0,C 180,E1 -15280.96,E2 -15280.96} C_VEL
LIN {X 0,Y 319.729,Z 248.659,A -85,B 0,C 180,E1 -15285.274,E2 -15285.274} C_VEL
LIN {X 0,Y 319.755,Z 248.655,A -85,B 0,C 180,E1 -15289.871,E2 -15289.871} C_VEL
LIN {X 0,Y 319.93,Z 248.635,A -85,B 0,C 180,E1 -15292.424,E2 -15292.424} C_VEL
LIN {X 0,Y 319.746,Z 248.658,A -85,B 0,C 180,E1 -15294.954,E2 -15294.954} C_VEL
LIN {X 0,Y 319.989,Z 248.625,A -85,B 0,C 180,E1 -15297.48,E2 -15297.48} C_VEL
LIN {X 0,Y 320.166,Z 248.604,A -85,B 0,C 180,E1 -15299.998,E2 -15299.998} C_VEL
LIN {X 0,Y 319.987,Z 248.627,A -85,B 0,C 180,E1 -15302.515,E2 -15302.515} C_VEL
LIN {X 0,Y 319.926,Z 248.634,A -85,B 0,C 180,E1 -15306.665,E2 -15306.665} C_VEL
LIN {X 0,Y 319.868,Z 248.816,A -85,B 0,C 180,E1 -15308.845,E2 -15308.845} C_VEL
LIN {X 0,Y 319.778,Z 251.304,A -85,B 0,C 180,E1 -15312.694,E2 -15312.694} C_VEL
LIN {X 0,Y 319.641,Z 253.1,A -85,B 0,C 180,E1 -15315.296,E2 -15315.296} C_VEL
LIN {X 0,Y 319.339,Z 255.994,A -85,B 0,C 180,E1 -15319.273,E2 -15319.273} C_VEL
LIN {X 0,Y 319.102,Z 259.158,A -85,B 0,C 180,E1 -15323.439,E2 -15323.439} C_VEL
LIN {X 0,Y 320.923,Z 264.326,A -85,B 0,C 180,E1 -15323.854,E2 -15323.854} C_VEL
LIN {X 0,Y 324.583,Z 275.051,A -85,B 0,C 180,E1 -15324.801,E2 -15324.801} C_VEL
LIN {X 0,Y 327.514,Z 286.48,A -85,B 0,C 180,E1 -15325.924,E2 -15325.924} C_VEL
LIN {X 0,Y 328.53,Z 292.055,A -85,B 0,C 180,E1 -15326.521,E2 -15326.521} C_VEL
LIN {X 0,Y 327.249,Z 303.232,A -85,B 0,C 180,E1 -15327.64,E2 -15327.64} C_VEL
LIN {X 0,Y 325.771,Z 314.269,A -85,B 0,C 180,E1 -15329.036,E2 -15329.036} C_VEL
LIN {X 0,Y 324.201,Z 324.451,A -85,B 0,C 180,E1 -15330.664,E2 -15330.664} C_VEL
LIN {X 0,Y 322.76,Z 333.362,A -85,B 0,C 180,E1 -15332.439,E2 -15332.439} C_VEL
LIN {X 0,Y 321.539,Z 340.55,A -85,B 0,C 180,E1 -15334.222,E2 -15334.222} C_VEL
LIN {X 0,Y 320.324,Z 347.242,A -85,B 0,C 180,E1 -15336.323,E2 -15336.323} C_VEL
LIN {X 0,Y 319.613,Z 351.443,A -85,B 0,C 180,E1 -15337.999,E2 -15337.999} C_VEL
LIN {X 0,Y 319.024,Z 354.824,A -85,B 0,C 180,E1 -15339.703,E2 -15339.703} C_VEL
LIN {X 0,Y 318.568,Z 357.393,A -85,B 0,C 180,E1 -15341.436,E2 -15341.436} C_VEL
LIN {X 0,Y 318.219,Z 359.173,A -85,B 0,C 180,E1 -15343.214,E2 -15343.214} C_VEL
LIN {X 0,Y 317.975,Z 360.166,A -85,B 0,C 180,E1 -15345.01,E2 -15345.01} C_VEL
LIN {X 0,Y 317.861,Z 360.357,A -85,B 0,C 180,E1 -15346.852,E2 -15346.852} C_VEL
LIN {X 0,Y 317.874,Z 359.682,A -85,B 0,C 180,E1 -15348.735,E2 -15348.735} C_VEL
LIN {X 0,Y 318.083,Z 358.072,A -85,B 0,C 180,E1 -15350.649,E2 -15350.649} C_VEL
LIN {X 0,Y 318.411,Z 355.415,A -85,B 0,C 180,E1 -15352.612,E2 -15352.612} C_VEL
LIN {X 0,Y 318.99,Z 350.572,A -85,B 0,C 180,E1 -15355.053,E2 -15355.053} C_VEL
LIN {X 0,Y 319.67,Z 345.151,A -85,B 0,C 180,E1 -15357.078,E2 -15357.078} C_VEL
LIN {X 0,Y 320.432,Z 339.351,A -85,B 0,C 180,E1 -15358.797,E2 -15358.797} C_VEL
LIN {X 0,Y 321.474,Z 331.326,A -85,B 0,C 180,E1 -15360.715,E2 -15360.715} C_VEL
LIN {X 0,Y 322.776,Z 321.313,A -85,B 0,C 180,E1 -15362.616,E2 -15362.616} C_VEL
LIN {X 0,Y 323.914,Z 311.503,A -85,B 0,C 180,E1 -15364.11,E2 -15364.11} C_VEL
LIN {X 0,Y 325.225,Z 299.825,A -85,B 0,C 180,E1 -15365.522,E2 -15365.522} C_VEL
LIN {X 0,Y 326.306,Z 287.745,A -85,B 0,C 180,E1 -15366.673,E2 -15366.673} C_VEL
LIN {X 0,Y 324.07,Z 277.063,A -85,B 0,C 180,E1 -15367.64,E2 -15367.64} C_VEL
LIN {X 0,Y 320.749,Z 264.12,A -85,B 0,C 180,E1 -15368.596,E2 -15368.596} C_VEL
LIN {X 0,Y 318.581,Z 256.321,A -85,B 0,C 180,E1 -15369.079,E2 -15369.079} C_VEL
LIN {X 0,Y 318.699,Z 253.648,A -85,B 0,C 180,E1 -15372.018,E2 -15372.018} C_VEL
LIN {X 0,Y 318.904,Z 250.132,A -85,B 0,C 180,E1 -15375.972,E2 -15375.972} C_VEL
LIN {X 0,Y 318.972,Z 249.015,A -85,B 0,C 180,E1 -15377.272,E2 -15377.272} C_VEL
LIN {X 0,Y 319.326,Z 248.707,A -85,B 0,C 180,E1 -15379.86,E2 -15379.86} C_VEL
LIN {X 0,Y 319.76,Z 248.651,A -85,B 0,C 180,E1 -15382.423,E2 -15382.423} C_VEL
LIN {X 0,Y 319.87,Z 248.641,A -85,B 0,C 180,E1 -15383.694,E2 -15383.694} C_VEL
LIN {X 0,Y 319.994,Z 248.626,A -85,B 0,C 180,E1 -15387.483,E2 -15387.483} C_VEL
LIN {X 0,Y 320.154,Z 248.603,A -85,B 0,C 180,E1 -15390.001,E2 -15390.001} C_VEL
LIN {X 0,Y 319.977,Z 248.625,A -85,B 0,C 180,E1 -15392.518,E2 -15392.518} C_VEL
LIN {X 0,Y 319.937,Z 248.629,A -85,B 0,C 180,E1 -15396.306,E2 -15396.306} C_VEL
LIN {X 0,Y 319.828,Z 248.646,A -85,B 0,C 180,E1 -15398.849,E2 -15398.849} C_VEL
LIN {X 0,Y 319.67,Z 248.664,A -85,B 0,C 180,E1 -15402.701,E2 -15402.701} C_VEL
LIN {X 0,Y 319.685,Z 248.664,A -85,B 0,C 180,E1 -15405.297,E2 -15405.297} C_VEL
LIN {X 0,Y 319.677,Z 248.664,A -85,B 0,C 180,E1 -15409.255,E2 -15409.255} C_VEL
LIN {X 0,Y 319.625,Z 248.67,A -85,B 0,C 180,E1 -15413.316,E2 -15413.316} C_VEL
LIN {X 0,Y 319.624,Z 248.668,A -85,B 0,C 180,E1 -15416.09,E2 -15416.09} C_VEL
LIN {X 0,Y 319.577,Z 248.678,A -85,B 0,C 180,E1 -15418.935,E2 -15418.935} C_VEL
LIN {X 0,Y 319.52,Z 248.681,A -85,B 0,C 180,E1 -15421.864,E2 -15421.864} C_VEL
LIN {X 0,Y 319.569,Z 248.675,A -85,B 0,C 180,E1 -15425.545,E2 -15425.545} C_VEL
LIN {X 0,Y 319.574,Z 248.675,A -85,B 0,C 180,E1 -15428.009,E2 -15428.009} C_VEL
LIN {X 0,Y 319.592,Z 248.672,A -85,B 0,C 180,E1 -15431.614,E2 -15431.614} C_VEL
LIN {X 0,Y 319.637,Z 248.666,A -85,B 0,C 180,E1 -15435.287,E2 -15435.287} C_VEL
LIN {X 0,Y 319.576,Z 248.677,A -85,B 0,C 180,E1 -15438.723,E2 -15438.723} C_VEL
LIN {X 0,Y 319.593,Z 248.677,A -85,B 0,C 180,E1 -15442.341,E2 -15442.341} C_VEL
LIN {X 0,Y 319.555,Z 248.677,A -85,B 0,C 180,E1 -15445.126,E2 -15445.126} C_VEL
LIN {X 0,Y 319.57,Z 248.674,A -85,B 0,C 180,E1 -15449.059,E2 -15449.059} C_VEL
LIN {X 0,Y 319.606,Z 248.673,A -85,B 0,C 180,E1 -15452.501,E2 -15452.501} C_VEL
LIN {X 0,Y 319.602,Z 248.671,A -85,B 0,C 180,E1 -15455.306,E2 -15455.306} C_VEL
LIN {X 0,Y 319.605,Z 248.671,A -85,B 0,C 180,E1 -15457.436,E2 -15457.436} C_VEL
LIN {X 0,Y 319.014,Z 248.749,A -85,B 0,C 180,E1 -15458.488,E2 -15458.488} C_VEL
LIN {X 0,Y 316.203,Z 249.101,A -85,B 0,C 180,E1 -15460.202,E2 -15460.202} C_VEL
LIN {X 0,Y 313.765,Z 249.402,A -85,B 0,C 180,E1 -15461.59,E2 -15461.59} C_VEL
LIN {X 0,Y 312.699,Z 249.531,A -85,B 0,C 180,E1 -15462.666,E2 -15462.666} C_VEL
LIN {X 0,Y 312.605,Z 249.541,A -85,B 0,C 180,E1 -15463.03,E2 -15463.03} C_VEL
LIN {X 0,Y 312.693,Z 249.533,A -85,B 0,C 180,E1 -15465.689,E2 -15465.689} C_VEL
LIN {X 0,Y 312.698,Z 249.534,A -85,B 0,C 180,E1 -15469.644,E2 -15469.644} C_VEL
LIN {X 0,Y 312.894,Z 249.509,A -85,B 0,C 180,E1 -15473.554,E2 -15473.554} C_VEL
LIN {X 0,Y 312.938,Z 249.502,A -85,B 0,C 180,E1 -15477.428,E2 -15477.428} C_VEL
LIN {X 0,Y 313.104,Z 249.484,A -85,B 0,C 180,E1 -15480.002,E2 -15480.002} C_VEL
LIN {X 0,Y 312.938,Z 249.501,A -85,B 0,C 180,E1 -15482.576,E2 -15482.576} C_VEL
LIN {X 0,Y 312.853,Z 249.51,A -85,B 0,C 180,E1 -15486.451,E2 -15486.451} C_VEL
LIN {X 0,Y 312.755,Z 249.524,A -85,B 0,C 180,E1 -15489.052,E2 -15489.052} C_VEL
LIN {X 0,Y 312.639,Z 249.539,A -85,B 0,C 180,E1 -15492.993,E2 -15492.993} C_VEL
LIN {X 0,Y 312.644,Z 249.541,A -85,B 0,C 180,E1 -15495.651,E2 -15495.651} C_VEL
LIN {X 0,Y 312.636,Z 249.542,A -85,B 0,C 180,E1 -15499.238,E2 -15499.238} C_VEL
LIN {X 0,Y 312.552,Z 249.55,A -85,B 0,C 180,E1 -15502.791,E2 -15502.791} C_VEL
LIN {X 0,Y 312.603,Z 249.544,A -85,B 0,C 180,E1 -15505.935,E2 -15505.935} C_VEL
LIN {X 0,Y 312.545,Z 249.552,A -85,B 0,C 180,E1 -15509.652,E2 -15509.652} C_VEL
LIN {X 0,Y 312.527,Z 249.554,A -85,B 0,C 180,E1 -15513.69,E2 -15513.69} C_VEL
LIN {X 0,Y 312.533,Z 249.556,A -85,B 0,C 180,E1 -15517.386,E2 -15517.386} C_VEL
LIN {X 0,Y 312.521,Z 249.564,A -85,B 0,C 180,E1 -15521.072,E2 -15521.072} C_VEL
LIN {X 0,Y 313.252,Z 253.565,A -85,B 0,C 180,E1 -15524.115,E2 -15524.115} C_VEL
LIN {X 0,Y 314.202,Z 258.766,A -85,B 0,C 180,E1 -15527.852,E2 -15527.852} C_VEL
LIN {X 0,Y 315.117,Z 263.94,A -85,B 0,C 180,E1 -15531.355,E2 -15531.355} C_VEL
LIN {X 0,Y 315.317,Z 267.084,A -85,B 0,C 180,E1 -15533.362,E2 -15533.362} C_VEL
LIN {X 0,Y 314.788,Z 271.554,A -85,B 0,C 180,E1 -15536.071,E2 -15536.071} C_VEL
LIN {X 0,Y 313.669,Z 279.093,A -85,B 0,C 180,E1 -15540.466,E2 -15540.466} C_VEL
LIN {X 0,Y 312.889,Z 285.226,A -85,B 0,C 180,E1 -15543.96,E2 -15543.96} C_VEL
LIN {X 0,Y 312.263,Z 290.935,A -85,B 0,C 180,E1 -15547.139,E2 -15547.139} C_VEL
LIN {X 0,Y 314.721,Z 304.953,A -85,B 0,C 180,E1 -15547.902,E2 -15547.902} C_VEL
LIN {X 0,Y 316.483,Z 318.025,A -85,B 0,C 180,E1 -15548.859,E2 -15548.859} C_VEL
LIN {X 0,Y 317.544,Z 329.806,A -85,B 0,C 180,E1 -15549.936,E2 -15549.936} C_VEL
LIN {X 0,Y 317.942,Z 336.338,A -85,B 0,C 180,E1 -15550.635,E2 -15550.635} C_VEL
LIN {X 0,Y 316.299,Z 348.068,A -85,B 0,C 180,E1 -15552.043,E2 -15552.043} C_VEL
LIN {X 0,Y 315.101,Z 358.048,A -85,B 0,C 180,E1 -15553.555,E2 -15553.555} C_VEL
LIN {X 0,Y 313.996,Z 366.307,A -85,B 0,C 180,E1 -15555.084,E2 -15555.084} C_VEL
LIN {X 0,Y 312.799,Z 374.771,A -85,B 0,C 180,E1 -15557.015,E2 -15557.015} C_VEL
LIN {X 0,Y 311.945,Z 381.582,A -85,B 0,C 180,E1 -15558.959,E2 -15558.959} C_VEL
LIN {X 0,Y 311.365,Z 387.025,A -85,B 0,C 180,E1 -15560.908,E2 -15560.908} C_VEL
LIN {X 0,Y 311.01,Z 391.268,A -85,B 0,C 180,E1 -15562.86,E2 -15562.86} C_VEL
LIN {X 0,Y 310.868,Z 394.429,A -85,B 0,C 180,E1 -15564.811,E2 -15564.811} C_VEL
LIN {X 0,Y 310.847,Z 395.993,A -85,B 0,C 180,E1 -15566.11,E2 -15566.11} C_VEL
LIN {X 0,Y 310.787,Z 397.114,A -85,B 0,C 180,E1 -15567.407,E2 -15567.407} C_VEL
LIN {X 0,Y 310.854,Z 397.804,A -85,B 0,C 180,E1 -15568.704,E2 -15568.704} C_VEL
LIN {X 0,Y 310.957,Z 398.099,A -85,B 0,C 180,E1 -15569.999,E2 -15569.999} C_VEL
LIN {X 0,Y 310.849,Z 397.984,A -85,B 0,C 180,E1 -15571.295,E2 -15571.295} C_VEL
LIN {X 0,Y 310.786,Z 397.457,A -85,B 0,C 180,E1 -15572.591,E2 -15572.591} C_VEL
LIN {X 0,Y 310.821,Z 396.501,A -85,B 0,C 180,E1 -15573.889,E2 -15573.889} C_VEL
LIN {X 0,Y 310.897,Z 394.195,A -85,B 0,C 180,E1 -15575.92,E2 -15575.92} C_VEL
LIN {X 0,Y 311.206,Z 389.857,A -85,B 0,C 180,E1 -15578.44,E2 -15578.44} C_VEL
LIN {X 0,Y 311.727,Z 385.266,A -85,B 0,C 180,E1 -15580.39,E2 -15580.39} C_VEL
LIN {X 0,Y 312.656,Z 378.373,A -85,B 0,C 180,E1 -15582.659,E2 -15582.659} C_VEL
LIN {X 0,Y 313.921,Z 370.943,A -85,B 0,C 180,E1 -15584.587,E2 -15584.587} C_VEL
LIN {X 0,Y 315.164,Z 362.858,A -85,B 0,C 180,E1 -15586.3,E2 -15586.3} C_VEL
LIN {X 0,Y 316.565,Z 353.412,A -85,B 0,C 180,E1 -15587.94,E2 -15587.94} C_VEL
LIN {X 0,Y 318.178,Z 343.277,A -85,B 0,C 180,E1 -15589.348,E2 -15589.348} C_VEL
LIN {X 0,Y 319.065,Z 336.625,A -85,B 0,C 180,E1 -15590.13,E2 -15590.13} C_VEL
LIN {X 0,Y 318.558,Z 324.734,A -85,B 0,C 180,E1 -15591.436,E2 -15591.436} C_VEL
LIN {X 0,Y 317.489,Z 312.955,A -85,B 0,C 180,E1 -15592.505,E2 -15592.505} C_VEL
LIN {X 0,Y 315.314,Z 300.583,A -85,B 0,C 180,E1 -15593.482,E2 -15593.482} C_VEL
LIN {X 0,Y 312.518,Z 288.842,A -85,B 0,C 180,E1 -15594.291,E2 -15594.291} C_VEL
LIN {X 0,Y 313.34,Z 282.239,A -85,B 0,C 180,E1 -15598.099,E2 -15598.099} C_VEL
LIN {X 0,Y 314.304,Z 276.039,A -85,B 0,C 180,E1 -15601.818,E2 -15601.818} C_VEL
LIN {X 0,Y 315.272,Z 270.352,A -85,B 0,C 180,E1 -15605.42,E2 -15605.42} C_VEL
LIN {X 0,Y 315.512,Z 266.89,A -85,B 0,C 180,E1 -15607.774,E2 -15607.774} C_VEL
LIN {X 0,Y 314.975,Z 263.056,A -85,B 0,C 180,E1 -15610.653,E2 -15610.653} C_VEL
LIN {X 0,Y 314.181,Z 258.653,A -85,B 0,C 180,E1 -15614.288,E2 -15614.288} C_VEL
LIN {X 0,Y 313.533,Z 254.927,A -85,B 0,C 180,E1 -15617.74,E2 -15617.74} C_VEL
LIN {X 0,Y 312.806,Z 251.163,A -85,B 0,C 180,E1 -15621.846,E2 -15621.846} C_VEL
LIN {X 0,Y 312.538,Z 249.558,A -85,B 0,C 180,E1 -15624.048,E2 -15624.048} C_VEL
LIN {X 0,Y 312.505,Z 249.558,A -85,B 0,C 180,E1 -15627.332,E2 -15627.332} C_VEL
LIN {X 0,Y 312.552,Z 249.551,A -85,B 0,C 180,E1 -15631.274,E2 -15631.274} C_VEL
LIN {X 0,Y 312.585,Z 249.549,A -85,B 0,C 180,E1 -15634.709,E2 -15634.709} C_VEL
LIN {X 0,Y 312.587,Z 249.544,A -85,B 0,C 180,E1 -15637.527,E2 -15637.527} C_VEL
LIN {X 0,Y 312.637,Z 249.539,A -85,B 0,C 180,E1 -15641.654,E2 -15641.654} C_VEL
LIN {X 0,Y 312.692,Z 249.537,A -85,B 0,C 180,E1 -15645.684,E2 -15645.684} C_VEL
LIN {X 0,Y 312.699,Z 249.532,A -85,B 0,C 180,E1 -15649.64,E2 -15649.64} C_VEL
LIN {X 0,Y 312.869,Z 249.514,A -85,B 0,C 180,E1 -15652.252,E2 -15652.252} C_VEL
LIN {X 0,Y 312.716,Z 249.534,A -85,B 0,C 180,E1 -15654.84,E2 -15654.84} C_VEL
LIN {X 0,Y 312.989,Z 249.5,A -85,B 0,C 180,E1 -15658.711,E2 -15658.711} C_VEL
LIN {X 0,Y 313.117,Z 249.482,A -85,B 0,C 180,E1 -15659.998,E2 -15659.998} C_VEL
LIN {X 0,Y 312.933,Z 249.505,A -85,B 0,C 180,E1 -15662.572,E2 -15662.572} C_VEL
LIN {X 0,Y 312.889,Z 249.511,A -85,B 0,C 180,E1 -15666.648,E2 -15666.648} C_VEL
LIN {X 0,Y 312.866,Z 249.515,A -85,B 0,C 180,E1 -15667.744,E2 -15667.744} C_VEL
LIN {X 0,Y 312.81,Z 251.025,A -85,B 0,C 180,E1 -15670.352,E2 -15670.352} C_VEL
LIN {X 0,Y 312.779,Z 252.691,A -85,B 0,C 180,E1 -15672.983,E2 -15672.983} C_VEL
LIN {X 0,Y 312.595,Z 254.503,A -85,B 0,C 180,E1 -15675.649,E2 -15675.649} C_VEL
LIN {X 0,Y 312.284,Z 257.415,A -85,B 0,C 180,E1 -15679.727,E2 -15679.727} C_VEL
LIN {X 0,Y 312.119,Z 259.673,A -85,B 0,C 180,E1 -15682.766,E2 -15682.766} C_VEL
LIN {X 0,Y 314.345,Z 265.752,A -85,B 0,C 180,E1 -15683.291,E2 -15683.291} C_VEL
LIN {X 0,Y 318.041,Z 276.576,A -85,B 0,C 180,E1 -15684.301,E2 -15684.301} C_VEL
LIN {X 0,Y 320.89,Z 287.678,A -85,B 0,C 180,E1 -15685.453,E2 -15685.453} C_VEL
LIN {X 0,Y 321.93,Z 293.574,A -85,B 0,C 180,E1 -15686.113,E2 -15686.113} C_VEL
LIN {X 0,Y 320.647,Z 304.291,A -85,B 0,C 180,E1 -15687.226,E2 -15687.226} C_VEL
LIN {X 0,Y 319.135,Z 314.928,A -85,B 0,C 180,E1 -15688.609,E2 -15688.609} C_VEL
LIN {X 0,Y 317.703,Z 323.919,A -85,B 0,C 180,E1 -15690.059,E2 -15690.059} C_VEL
LIN {X 0,Y 316.151,Z 332.929,A -85,B 0,C 180,E1 -15691.853,E2 -15691.853} C_VEL
LIN {X 0,Y 314.639,Z 341.254,A -85,B 0,C 180,E1 -15693.943,E2 -15693.943} C_VEL
LIN {X 0,Y 313.342,Z 348.057,A -85,B 0,C 180,E1 -15696.154,E2 -15696.154} C_VEL
LIN {X 0,Y 312.519,Z 352.646,A -85,B 0,C 180,E1 -15698.087,E2 -15698.087} C_VEL
LIN {X 0,Y 311.887,Z 356.088,A -85,B 0,C 180,E1 -15699.992,E2 -15699.992} C_VEL
LIN {X 0,Y 311.237,Z 359.273,A -85,B 0,C 180,E1 -15702.639,E2 -15702.639} C_VEL
LIN {X 0,Y 310.956,Z 360.472,A -85,B 0,C 180,E1 -15704.474,E2 -15704.474} C_VEL
LIN {X 0,Y 310.785,Z 360.842,A -85,B 0,C 180,E1 -15706.352,E2 -15706.352} C_VEL
LIN {X 0,Y 310.82,Z 359.902,A -85,B 0,C 180,E1 -15709.027,E2 -15709.027} C_VEL
LIN {X 0,Y 311.006,Z 358.407,A -85,B 0,C 180,E1 -15710.749,E2 -15710.749} C_VEL
LIN {X 0,Y 311.478,Z 354.817,A -85,B 0,C 180,E1 -15713.279,E2 -15713.279} C_VEL
LIN {X 0,Y 312.128,Z 349.637,A -85,B 0,C 180,E1 -15715.744,E2 -15715.744} C_VEL
LIN {X 0,Y 312.922,Z 343.263,A -85,B 0,C 180,E1 -15717.982,E2 -15717.982} C_VEL
LIN {X 0,Y 313.817,Z 336.924,A -85,B 0,C 180,E1 -15719.743,E2 -15719.743} C_VEL
LIN {X 0,Y 315.014,Z 328.187,A -85,B 0,C 180,E1 -15721.701,E2 -15721.701} C_VEL
LIN {X 0,Y 316.285,Z 318.457,A -85,B 0,C 180,E1 -15723.441,E2 -15723.441} C_VEL
LIN {X 0,Y 317.576,Z 307.765,A -85,B 0,C 180,E1 -15724.979,E2 -15724.979} C_VEL
LIN {X 0,Y 318.785,Z 296.351,A -85,B 0,C 180,E1 -15726.276,E2 -15726.276} C_VEL
LIN {X 0,Y 319.409,Z 288.564,A -85,B 0,C 180,E1 -15727.012,E2 -15727.012} C_VEL
LIN {X 0,Y 317.077,Z 277.575,A -85,B 0,C 180,E1 -15728.036,E2 -15728.036} C_VEL
LIN {X 0,Y 313.681,Z 264.375,A -85,B 0,C 180,E1 -15729.037,E2 -15729.037} C_VEL
LIN {X 0,Y 311.518,Z 256.713,A -85,B 0,C 180,E1 -15729.533,E2 -15729.533} C_VEL
LIN {X 0,Y 311.664,Z 253.653,A -85,B 0,C 180,E1 -15732.954,E2 -15732.954} C_VEL
LIN {X 0,Y 311.904,Z 250.152,A -85,B 0,C 180,E1 -15736.979,E2 -15736.979} C_VEL
LIN {X 0,Y 312.04,Z 249.62,A -85,B 0,C 180,E1 -15738.306,E2 -15738.306} C_VEL
LIN {X 0,Y 312.685,Z 249.533,A -85,B 0,C 180,E1 -15742.25,E2 -15742.25} C_VEL
LIN {X 0,Y 312.691,Z 249.534,A -85,B 0,C 180,E1 -15744.843,E2 -15744.843} C_VEL
LIN {X 0,Y 312.937,Z 249.506,A -85,B 0,C 180,E1 -15747.426,E2 -15747.426} C_VEL
LIN {X 0,Y 313.106,Z 249.481,A -85,B 0,C 180,E1 -15750.001,E2 -15750.001} C_VEL
LIN {X 0,Y 312.924,Z 249.504,A -85,B 0,C 180,E1 -15752.575,E2 -15752.575} C_VEL
LIN {X 0,Y 312.896,Z 249.507,A -85,B 0,C 180,E1 -15756.449,E2 -15756.449} C_VEL
LIN {X 0,Y 312.773,Z 249.527,A -85,B 0,C 180,E1 -15759.05,E2 -15759.05} C_VEL
LIN {X 0,Y 312.623,Z 249.545,A -85,B 0,C 180,E1 -15762.992,E2 -15762.992} C_VEL
LIN {X 0,Y 312.624,Z 249.541,A -85,B 0,C 180,E1 -15765.651,E2 -15765.651} C_VEL
LIN {X 0,Y 312.621,Z 249.541,A -85,B 0,C 180,E1 -15769.708,E2 -15769.708} C_VEL
LIN {X 0,Y 312.572,Z 249.547,A -85,B 0,C 180,E1 -15773.874,E2 -15773.874} C_VEL
LIN {X 0,Y 312.571,Z 249.551,A -85,B 0,C 180,E1 -15776.724,E2 -15776.724} C_VEL
LIN {X 0,Y 312.533,Z 249.552,A -85,B 0,C 180,E1 -15779.652,E2 -15779.652} C_VEL
LIN {X 0,Y 312.508,Z 249.555,A -85,B 0,C 180,E1 -15783.691,E2 -15783.691} C_VEL
LIN {X 0,Y 312.531,Z 249.551,A -85,B 0,C 180,E1 -15787.385,E2 -15787.385} C_VEL
LIN {X 0,Y 312.518,Z 249.558,A -85,B 0,C 180,E1 -15790.705,E2 -15790.705} C_VEL
LIN {X 0,Y 312.586,Z 249.547,A -85,B 0,C 180,E1 -15794.186,E2 -15794.186} C_VEL
LIN {X 0,Y 312.549,Z 249.549,A -85,B 0,C 180,E1 -15797.906,E2 -15797.906} C_VEL
LIN {X 0,Y 312.552,Z 249.55,A -85,B 0,C 180,E1 -15801.907,E2 -15801.907} C_VEL
LIN {X 0,Y 312.501,Z 249.556,A -85,B 0,C 180,E1 -15805.793,E2 -15805.793} C_VEL
LIN {X 0,Y 312.524,Z 249.552,A -85,B 0,C 180,E1 -15808.857,E2 -15808.857} C_VEL
LIN {X 0,Y 312.571,Z 249.548,A -85,B 0,C 180,E1 -15811.827,E2 -15811.827} C_VEL
LIN {X 0,Y 312.582,Z 249.547,A -85,B 0,C 180,E1 -15814.713,E2 -15814.713} C_VEL
LIN {X 0,Y 312.585,Z 249.546,A -85,B 0,C 180,E1 -15817.531,E2 -15817.531} C_VEL
LIN {X 0,Y 312.637,Z 249.539,A -85,B 0,C 180,E1 -15821.659,E2 -15821.659} C_VEL
LIN {X 0,Y 312.605,Z 249.541,A -85,B 0,C 180,E1 -15823.03,E2 -15823.03} C_VEL
LIN {X 0,Y 311.916,Z 249.632,A -85,B 0,C 180,E1 -15824.106,E2 -15824.106} C_VEL
LIN {X 0,Y 309.065,Z 249.987,A -85,B 0,C 180,E1 -15825.859,E2 -15825.859} C_VEL
LIN {X 0,Y 306.675,Z 250.285,A -85,B 0,C 180,E1 -15827.279,E2 -15827.279} C_VEL
LIN {X 0,Y 305.671,Z 250.409,A -85,B 0,C 180,E1 -15828.379,E2 -15828.379} C_VEL
LIN {X 0,Y 305.599,Z 250.416,A -85,B 0,C 180,E1 -15828.752,E2 -15828.752} C_VEL
LIN {X 0,Y 305.773,Z 250.396,A -85,B 0,C 180,E1 -15832.076,E2 -15832.076} C_VEL
LIN {X 0,Y 305.685,Z 250.402,A -85,B 0,C 180,E1 -15834.726,E2 -15834.726} C_VEL
LIN {X 0,Y 305.96,Z 250.37,A -85,B 0,C 180,E1 -15838.686,E2 -15838.686} C_VEL
LIN {X 0,Y 305.958,Z 250.372,A -85,B 0,C 180,E1 -15841.318,E2 -15841.318} C_VEL
LIN {X 0,Y 305.676,Z 250.407,A -85,B 0,C 180,E1 -15845.279,E2 -15845.279} C_VEL
LIN {X 0,Y 305.765,Z 250.397,A -85,B 0,C 180,E1 -15847.929,E2 -15847.929} C_VEL
LIN {X 0,Y 305.603,Z 250.417,A -85,B 0,C 180,E1 -15851.947,E2 -15851.947} C_VEL
LIN {X 0,Y 305.644,Z 250.411,A -85,B 0,C 180,E1 -15855.037,E2 -15855.037} C_VEL
LIN {X 0,Y 305.582,Z 250.423,A -85,B 0,C 180,E1 -15859.446,E2 -15859.446} C_VEL
LIN {X 0,Y 305.497,Z 250.431,A -85,B 0,C 180,E1 -15863.043,E2 -15863.043} C_VEL
LIN {X 0,Y 305.532,Z 250.424,A -85,B 0,C 180,E1 -15866.22,E2 -15866.22} C_VEL
LIN {X 0,Y 305.495,Z 250.432,A -85,B 0,C 180,E1 -15869.049,E2 -15869.049} C_VEL
LIN {X 0,Y 305.449,Z 250.435,A -85,B 0,C 180,E1 -15871.954,E2 -15871.954} C_VEL
LIN {X 0,Y 305.47,Z 250.437,A -85,B 0,C 180,E1 -15875.114,E2 -15875.114} C_VEL
LIN {X 0,Y 305.456,Z 250.437,A -85,B 0,C 180,E1 -15878.53,E2 -15878.53} C_VEL
LIN {X 0,Y 305.496,Z 250.497,A -85,B 0,C 180,E1 -15880.701,E2 -15880.701} C_VEL
LIN {X 0,Y 306.148,Z 254.081,A -85,B 0,C 180,E1 -15883.528,E2 -15883.528} C_VEL
LIN {X 0,Y 307.003,Z 258.934,A -85,B 0,C 180,E1 -15887.103,E2 -15887.103} C_VEL
LIN {X 0,Y 307.839,Z 263.435,A -85,B 0,C 180,E1 -15890.264,E2 -15890.264} C_VEL
LIN {X 0,Y 308.299,Z 267.449,A -85,B 0,C 180,E1 -15892.929,E2 -15892.929} C_VEL
LIN {X 0,Y 307.752,Z 272.358,A -85,B 0,C 180,E1 -15895.999,E2 -15895.999} C_VEL
LIN {X 0,Y 306.772,Z 278.606,A -85,B 0,C 180,E1 -15899.734,E2 -15899.734} C_VEL
LIN {X 0,Y 305.768,Z 286.092,A -85,B 0,C 180,E1 -15904.105,E2 -15904.105} C_VEL
LIN {X 0,Y 305.266,Z 290.578,A -85,B 0,C 180,E1 -15906.668,E2 -15906.668} C_VEL
LIN {X 0,Y 307.738,Z 304.646,A -85,B 0,C 180,E1 -15907.457,E2 -15907.457} C_VEL
LIN {X 0,Y 309.448,Z 317.38,A -85,B 0,C 180,E1 -15908.408,E2 -15908.408} C_VEL
LIN {X 0,Y 310.523,Z 329.095,A -85,B 0,C 180,E1 -15909.504,E2 -15909.504} C_VEL
LIN {X 0,Y 311.028,Z 336.795,A -85,B 0,C 180,E1 -15910.359,E2 -15910.359} C_VEL
LIN {X 0,Y 309.341,Z 348.363,A -85,B 0,C 180,E1 -15911.796,E2 -15911.796} C_VEL
LIN {X 0,Y 308.104,Z 358.261,A -85,B 0,C 180,E1 -15913.348,E2 -15913.348} C_VEL
LIN {X 0,Y 306.847,Z 367.123,A -85,B 0,C 180,E1 -15915.068,E2 -15915.068} C_VEL
LIN {X 0,Y 305.672,Z 375.35,A -85,B 0,C 180,E1 -15917.045,E2 -15917.045} C_VEL
LIN {X 0,Y 304.911,Z 380.962,A -85,B 0,C 180,E1 -15918.701,E2 -15918.701} C_VEL
LIN {X 0,Y 304.311,Z 386.446,A -85,B 0,C 180,E1 -15920.696,E2 -15920.696} C_VEL
LIN {X 0,Y 303.94,Z 390.725,A -85,B 0,C 180,E1 -15922.693,E2 -15922.693} C_VEL
LIN {X 0,Y 303.787,Z 393.92,A -85,B 0,C 180,E1 -15924.69,E2 -15924.69} C_VEL
LIN {X 0,Y 303.779,Z 395.501,A -85,B 0,C 180,E1 -15926.019,E2 -15926.019} C_VEL
LIN {X 0,Y 303.709,Z 396.65,A -85,B 0,C 180,E1 -15927.347,E2 -15927.347} C_VEL
LIN {X 0,Y 303.763,Z 397.355,A -85,B 0,C 180,E1 -15928.674,E2 -15928.674} C_VEL
LIN {X 0,Y 303.869,Z 397.663,A -85,B 0,C 180,E1 -15929.999,E2 -15929.999} C_VEL
LIN {X 0,Y 303.757,Z 397.562,A -85,B 0,C 180,E1 -15931.325,E2 -15931.325} C_VEL
LIN {X 0,Y 303.707,Z 397.06,A -85,B 0,C 180,E1 -15932.652,E2 -15932.652} C_VEL
LIN {X 0,Y 303.732,Z 396.119,A -85,B 0,C 180,E1 -15933.98,E2 -15933.98} C_VEL
LIN {X 0,Y 303.825,Z 394.051,A -85,B 0,C 180,E1 -15935.908,E2 -15935.908} C_VEL
LIN {X 0,Y 304.021,Z 390.825,A -85,B 0,C 180,E1 -15937.972,E2 -15937.972} C_VEL
LIN {X 0,Y 304.485,Z 386.649,A -85,B 0,C 180,E1 -15939.968,E2 -15939.968} C_VEL
LIN {X 0,Y 305.358,Z 380.294,A -85,B 0,C 180,E1 -15942.291,E2 -15942.291} C_VEL
LIN {X 0,Y 306.562,Z 373.434,A -85,B 0,C 180,E1 -15944.266,E2 -15944.266} C_VEL
LIN {X 0,Y 307.988,Z 364.999,A -85,B 0,C 180,E1 -15946.226,E2 -15946.226} C_VEL
LIN {X 0,Y 309.291,Z 356.325,A -85,B 0,C 180,E1 -15947.863,E2 -15947.863} C_VEL
LIN {X 0,Y 311.093,Z 345.767,A -85,B 0,C 180,E1 -15949.464,E2 -15949.464} C_VEL
LIN {X 0,Y 312.263,Z 338.208,A -85,B 0,C 180,E1 -15950.416,E2 -15950.416} C_VEL
LIN {X 0,Y 311.902,Z 325.596,A -85,B 0,C 180,E1 -15951.873,E2 -15951.873} C_VEL
LIN {X 0,Y 310.959,Z 314.032,A -85,B 0,C 180,E1 -15952.99,E2 -15952.99} C_VEL
LIN {X 0,Y 308.8,Z 301.688,A -85,B 0,C 180,E1 -15954.03,E2 -15954.03} C_VEL
LIN {X 0,Y 305.616,Z 288.367,A -85,B 0,C 180,E1 -15954.995,E2 -15954.995} C_VEL
LIN {X 0,Y 306.637,Z 280.947,A -85,B 0,C 180,E1 -15959.428,E2 -15959.428} C_VEL
LIN {X 0,Y 307.607,Z 274.871,A -85,B 0,C 180,E1 -15963.252,E2 -15963.252} C_VEL
LIN {X 0,Y 308.422,Z 270.218,A -85,B 0,C 180,E1 -15966.331,E2 -15966.331} C_VEL
LIN {X 0,Y 308.515,Z 267.929,A -85,B 0,C 180,E1 -15967.955,E2 -15967.955} C_VEL
LIN {X 0,Y 308.263,Z 265.675,A -85,B 0,C 180,E1 -15969.669,E2 -15969.669} C_VEL
LIN {X 0,Y 307.439,Z 261.277,A -85,B 0,C 180,E1 -15973.297,E2 -15973.297} C_VEL
LIN {X 0,Y 306.667,Z 257.076,A -85,B 0,C 180,E1 -15977.167,E2 -15977.167} C_VEL
LIN {X 0,Y 306.189,Z 254.386,A -85,B 0,C 180,E1 -15980.005,E2 -15980.005} C_VEL
LIN {X 0,Y 305.657,Z 251.422,A -85,B 0,C 180,E1 -15983.585,E2 -15983.585} C_VEL
LIN {X 0,Y 305.463,Z 250.435,A -85,B 0,C 180,E1 -15985.174,E2 -15985.174} C_VEL
LIN {X 0,Y 305.464,Z 250.436,A -85,B 0,C 180,E1 -15989.589,E2 -15989.589} C_VEL
LIN {X 0,Y 305.521,Z 250.429,A -85,B 0,C 180,E1 -15992.607,E2 -15992.607} C_VEL
LIN {X 0,Y 305.508,Z 250.43,A -85,B 0,C 180,E1 -15995.537,E2 -15995.537} C_VEL
LIN {X 0,Y 305.519,Z 250.424,A -85,B 0,C 180,E1 -15999.813,E2 -15999.813} C_VEL
LIN {X 0,Y 305.573,Z 250.418,A -85,B 0,C 180,E1 -16002.601,E2 -16002.601} C_VEL
LIN {X 0,Y 305.647,Z 250.413,A -85,B 0,C 180,E1 -16005.347,E2 -16005.347} C_VEL
LIN {X 0,Y 305.636,Z 250.411,A -85,B 0,C 180,E1 -16009.398,E2 -16009.398} C_VEL
LIN {X 0,Y 305.81,Z 250.391,A -85,B 0,C 180,E1 -16012.072,E2 -16012.072} C_VEL
LIN {X 0,Y 305.687,Z 250.409,A -85,B 0,C 180,E1 -16014.721,E2 -16014.721} C_VEL
LIN {X 0,Y 305.956,Z 250.376,A -85,B 0,C 180,E1 -16018.682,E2 -16018.682} C_VEL
LIN {X 0,Y 305.955,Z 250.374,A -85,B 0,C 180,E1 -16021.314,E2 -16021.314} C_VEL
LIN {X 0,Y 305.847,Z 250.389,A -85,B 0,C 180,E1 -16026.595,E2 -16026.595} C_VEL
LIN {X 0,Y 305.887,Z 251.619,A -85,B 0,C 180,E1 -16029.253,E2 -16029.253} C_VEL
LIN {X 0,Y 305.751,Z 254.109,A -85,B 0,C 180,E1 -16033.286,E2 -16033.286} C_VEL
LIN {X 0,Y 305.537,Z 255.924,A -85,B 0,C 180,E1 -16036.021,E2 -16036.021} C_VEL
LIN {X 0,Y 305.315,Z 258.223,A -85,B 0,C 180,E1 -16039.308,E2 -16039.308} C_VEL
LIN {X 0,Y 305.12,Z 260.234,A -85,B 0,C 180,E1 -16042.067,E2 -16042.067} C_VEL
LIN {X 0,Y 306.27,Z 263.394,A -85,B 0,C 180,E1 -16042.339,E2 -16042.339} C_VEL
LIN {X 0,Y 310.619,Z 275.194,A -85,B 0,C 180,E1 -16043.483,E2 -16043.483} C_VEL
LIN {X 0,Y 313.723,Z 286.316,A -85,B 0,C 180,E1 -16044.657,E2 -16044.657} C_VEL
LIN {X 0,Y 315.389,Z 294.948,A -85,B 0,C 180,E1 -16045.664,E2 -16045.664} C_VEL
LIN {X 0,Y 314.086,Z 305.152,A -85,B 0,C 180,E1 -16046.761,E2 -16046.761} C_VEL
LIN {X 0,Y 312.509,Z 315.706,A -85,B 0,C 180,E1 -16048.179,E2 -16048.179} C_VEL
LIN {X 0,Y 310.826,Z 325.549,A -85,B 0,C 180,E1 -16049.828,E2 -16049.828} C_VEL
LIN {X 0,Y 309.138,Z 334.814,A -85,B 0,C 180,E1 -16051.764,E2 -16051.764} C_VEL
LIN {X 0,Y 307.632,Z 342.717,A -85,B 0,C 180,E1 -16053.877,E2 -16053.877} C_VEL
LIN {X 0,Y 306.311,Z 349.269,A -85,B 0,C 180,E1 -16056.117,E2 -16056.117} C_VEL
LIN {X 0,Y 305.309,Z 354.423,A -85,B 0,C 180,E1 -16058.497,E2 -16058.497} C_VEL
LIN {X 0,Y 304.687,Z 357.494,A -85,B 0,C 180,E1 -16060.432,E2 -16060.432} C_VEL
LIN {X 0,Y 304.213,Z 359.607,A -85,B 0,C 180,E1 -16062.332,E2 -16062.332} C_VEL
LIN {X 0,Y 303.909,Z 360.85,A -85,B 0,C 180,E1 -16064.203,E2 -16064.203} C_VEL
LIN {X 0,Y 303.715,Z 361.266,A -85,B 0,C 180,E1 -16066.037,E2 -16066.037} C_VEL
LIN {X 0,Y 303.684,Z 360.941,A -85,B 0,C 180,E1 -16067.847,E2 -16067.847} C_VEL
LIN {X 0,Y 303.822,Z 359.793,A -85,B 0,C 180,E1 -16069.756,E2 -16069.756} C_VEL
LIN {X 0,Y 304.085,Z 357.623,A -85,B 0,C 180,E1 -16071.791,E2 -16071.791} C_VEL
LIN {X 0,Y 304.52,Z 354.332,A -85,B 0,C 180,E1 -16073.873,E2 -16073.873} C_VEL
LIN {X 0,Y 305.128,Z 349.727,A -85,B 0,C 180,E1 -16076.01,E2 -16076.01} C_VEL
LIN {X 0,Y 305.935,Z 343.561,A -85,B 0,C 180,E1 -16078.203,E2 -16078.203} C_VEL
LIN {X 0,Y 306.952,Z 336.735,A -85,B 0,C 180,E1 -16080.122,E2 -16080.122} C_VEL
LIN {X 0,Y 308.139,Z 328.187,A -85,B 0,C 180,E1 -16082.047,E2 -16082.047} C_VEL
LIN {X 0,Y 309.528,Z 317.899,A -85,B 0,C 180,E1 -16083.902,E2 -16083.902} C_VEL
LIN {X 0,Y 310.873,Z 306.917,A -85,B 0,C 180,E1 -16085.472,E2 -16085.472} C_VEL
LIN {X 0,Y 312.147,Z 295.196,A -85,B 0,C 180,E1 -16086.797,E2 -16086.797} C_VEL
LIN {X 0,Y 312.518,Z 289.437,A -85,B 0,C 180,E1 -16087.351,E2 -16087.351} C_VEL
LIN {X 0,Y 310.222,Z 278.643,A -85,B 0,C 180,E1 -16088.4,E2 -16088.4} C_VEL
LIN {X 0,Y 306.897,Z 265.628,A -85,B 0,C 180,E1 -16089.429,E2 -16089.429} C_VEL
LIN {X 0,Y 304.481,Z 257.123,A -85,B 0,C 180,E1 -16089.986,E2 -16089.986} C_VEL
LIN {X 0,Y 304.639,Z 253.663,A -85,B 0,C 180,E1 -16093.929,E2 -16093.929} C_VEL
LIN {X 0,Y 304.825,Z 251.314,A -85,B 0,C 180,E1 -16096.671,E2 -16096.671} C_VEL
LIN {X 0,Y 304.937,Z 250.505,A -85,B 0,C 180,E1 -16098.029,E2 -16098.029} C_VEL
LIN {X 0,Y 305.608,Z 250.415,A -85,B 0,C 180,E1 -16102.07,E2 -16102.07} C_VEL
LIN {X 0,Y 305.657,Z 250.41,A -85,B 0,C 180,E1 -16104.724,E2 -16104.724} C_VEL
LIN {X 0,Y 305.948,Z 250.373,A -85,B 0,C 180,E1 -16108.684,E2 -16108.684} C_VEL
LIN {X 0,Y 305.944,Z 250.377,A -85,B 0,C 180,E1 -16111.317,E2 -16111.317} C_VEL
LIN {X 0,Y 305.838,Z 250.386,A -85,B 0,C 180,E1 -16116.598,E2 -16116.598} C_VEL
LIN {X 0,Y 305.721,Z 250.404,A -85,B 0,C 180,E1 -16119.261,E2 -16119.261} C_VEL
LIN {X 0,Y 305.577,Z 250.422,A -85,B 0,C 180,E1 -16123.297,E2 -16123.297} C_VEL
LIN {X 0,Y 305.58,Z 250.418,A -85,B 0,C 180,E1 -16126.021,E2 -16126.021} C_VEL
LIN {X 0,Y 305.601,Z 250.417,A -85,B 0,C 180,E1 -16129.466,E2 -16129.466} C_VEL
LIN {X 0,Y 305.543,Z 250.427,A -85,B 0,C 180,E1 -16133.072,E2 -16133.072} C_VEL
LIN {X 0,Y 305.543,Z 250.423,A -85,B 0,C 180,E1 -16136.232,E2 -16136.232} C_VEL
LIN {X 0,Y 305.484,Z 250.433,A -85,B 0,C 180,E1 -16139.052,E2 -16139.052} C_VEL
LIN {X 0,Y 305.454,Z 250.434,A -85,B 0,C 180,E1 -16143.519,E2 -16143.519} C_VEL
LIN {X 0,Y 305.487,Z 250.433,A -85,B 0,C 180,E1 -16146.738,E2 -16146.738} C_VEL
LIN {X 0,Y 305.477,Z 250.436,A -85,B 0,C 180,E1 -16150.609,E2 -16150.609} C_VEL
LIN {X 0,Y 305.536,Z 250.428,A -85,B 0,C 180,E1 -16154.519,E2 -16154.519} C_VEL
LIN {X 0,Y 305.494,Z 250.428,A -85,B 0,C 180,E1 -16158.156,E2 -16158.156} C_VEL
LIN {X 0,Y 305.514,Z 250.426,A -85,B 0,C 180,E1 -16161.607,E2 -16161.607} C_VEL
LIN {X 0,Y 305.457,Z 250.434,A -85,B 0,C 180,E1 -16164.889,E2 -16164.889} C_VEL
LIN {X 0,Y 305.452,Z 250.436,A -85,B 0,C 180,E1 -16168.356,E2 -16168.356} C_VEL
LIN {X 0,Y 305.517,Z 250.424,A -85,B 0,C 180,E1 -16171.116,E2 -16171.116} C_VEL
LIN {X 0,Y 305.568,Z 250.423,A -85,B 0,C 180,E1 -16174.091,E2 -16174.091} C_VEL
LIN {X 0,Y 305.498,Z 250.43,A -85,B 0,C 180,E1 -16178.405,E2 -16178.405} C_VEL
LIN {X 0,Y 305.589,Z 250.415,A -85,B 0,C 180,E1 -16181.22,E2 -16181.22} C_VEL
LIN {X 0,Y 305.649,Z 250.409,A -85,B 0,C 180,E1 -16185.351,E2 -16185.351} C_VEL
LIN {X 0,Y 305.599,Z 250.416,A -85,B 0,C 180,E1 -16188.752,E2 -16188.752} C_VEL
LIN {X 0,Y 304.984,Z 250.497,A -85,B 0,C 180,E1 -16189.852,E2 -16189.852} C_VEL
LIN {X 0,Y 302.234,Z 250.837,A -85,B 0,C 180,E1 -16191.647,E2 -16191.647} C_VEL
LIN {X 0,Y 299.847,Z 251.134,A -85,B 0,C 180,E1 -16193.102,E2 -16193.102} C_VEL
LIN {X 0,Y 298.77,Z 251.266,A -85,B 0,C 180,E1 -16194.227,E2 -16194.227} C_VEL
LIN {X 0,Y 298.655,Z 251.278,A -85,B 0,C 180,E1 -16194.609,E2 -16194.609} C_VEL
LIN {X 0,Y 298.926,Z 251.246,A -85,B 0,C 180,E1 -16198.655,E2 -16198.655} C_VEL
LIN {X 0,Y 298.925,Z 251.249,A -85,B 0,C 180,E1 -16201.349,E2 -16201.349} C_VEL
LIN {X 0,Y 298.645,Z 251.284,A -85,B 0,C 180,E1 -16205.404,E2 -16205.404} C_VEL
LIN {X 0,Y 298.714,Z 251.273,A -85,B 0,C 180,E1 -16208.117,E2 -16208.117} C_VEL
LIN {X 0,Y 298.555,Z 251.293,A -85,B 0,C 180,E1 -16212.234,E2 -16212.234} C_VEL
LIN {X 0,Y 298.612,Z 251.288,A -85,B 0,C 180,E1 -16215.211,E2 -16215.211} C_VEL
LIN {X 0,Y 298.545,Z 251.297,A -85,B 0,C 180,E1 -16219.245,E2 -16219.245} C_VEL
LIN {X 0,Y 298.464,Z 251.308,A -85,B 0,C 180,E1 -16223.599,E2 -16223.599} C_VEL
LIN {X 0,Y 298.492,Z 251.301,A -85,B 0,C 180,E1 -16226.576,E2 -16226.576} C_VEL
LIN {X 0,Y 298.424,Z 251.312,A -85,B 0,C 180,E1 -16229.643,E2 -16229.643} C_VEL
LIN {X 0,Y 298.402,Z 251.314,A -85,B 0,C 180,E1 -16232.801,E2 -16232.801} C_VEL
LIN {X 0,Y 298.454,Z 251.309,A -85,B 0,C 180,E1 -16236.809,E2 -16236.809} C_VEL
LIN {X 0,Y 298.443,Z 251.438,A -85,B 0,C 180,E1 -16240.327,E2 -16240.327} C_VEL
LIN {X 0,Y 299.13,Z 255.066,A -85,B 0,C 180,E1 -16243.252,E2 -16243.252} C_VEL
LIN {X 0,Y 300.05,Z 260.292,A -85,B 0,C 180,E1 -16247.213,E2 -16247.213} C_VEL
LIN {X 0,Y 300.883,Z 264.788,A -85,B 0,C 180,E1 -16250.429,E2 -16250.429} C_VEL
LIN {X 0,Y 301.246,Z 268.052,A -85,B 0,C 180,E1 -16252.657,E2 -16252.657} C_VEL
LIN {X 0,Y 300.979,Z 271.39,A -85,B 0,C 180,E1 -16254.815,E2 -16254.815} C_VEL
LIN {X 0,Y 299.872,Z 278.091,A -85,B 0,C 180,E1 -16258.961,E2 -16258.961} C_VEL
LIN {X 0,Y 298.869,Z 285.344,A -85,B 0,C 180,E1 -16263.33,E2 -16263.33} C_VEL
LIN {X 0,Y 298.272,Z 290.211,A -85,B 0,C 180,E1 -16266.189,E2 -16266.189} C_VEL
LIN {X 0,Y 300.696,Z 304.101,A -85,B 0,C 180,E1 -16266.984,E2 -16266.984} C_VEL
LIN {X 0,Y 302.526,Z 317.666,A -85,B 0,C 180,E1 -16268.034,E2 -16268.034} C_VEL
LIN {X 0,Y 303.564,Z 328.633,A -85,B 0,C 180,E1 -16269.091,E2 -16269.091} C_VEL
LIN {X 0,Y 304.102,Z 337.189,A -85,B 0,C 180,E1 -16270.069,E2 -16270.069} C_VEL
LIN {X 0,Y 302.389,Z 348.617,A -85,B 0,C 180,E1 -16271.538,E2 -16271.538} C_VEL
LIN {X 0,Y 301.134,Z 358.336,A -85,B 0,C 180,E1 -16273.117,E2 -16273.117} C_VEL
LIN {X 0,Y 299.698,Z 367.887,A -85,B 0,C 180,E1 -16275.051,E2 -16275.051} C_VEL
LIN {X 0,Y 298.523,Z 375.915,A -85,B 0,C 180,E1 -16277.076,E2 -16277.076} C_VEL
LIN {X 0,Y 297.687,Z 382.349,A -85,B 0,C 180,E1 -16279.112,E2 -16279.112} C_VEL
LIN {X 0,Y 297.101,Z 387.446,A -85,B 0,C 180,E1 -16281.154,E2 -16281.154} C_VEL
LIN {X 0,Y 296.798,Z 391.39,A -85,B 0,C 180,E1 -16283.2,E2 -16283.2} C_VEL
LIN {X 0,Y 296.705,Z 393.409,A -85,B 0,C 180,E1 -16284.562,E2 -16284.562} C_VEL
LIN {X 0,Y 296.691,Z 395.006,A -85,B 0,C 180,E1 -16285.924,E2 -16285.924} C_VEL
LIN {X 0,Y 296.634,Z 396.18,A -85,B 0,C 180,E1 -16287.283,E2 -16287.283} C_VEL
LIN {X 0,Y 296.671,Z 396.905,A -85,B 0,C 180,E1 -16288.642,E2 -16288.642} C_VEL
LIN {X 0,Y 296.78,Z 397.227,A -85,B 0,C 180,E1 -16289.999,E2 -16289.999} C_VEL
LIN {X 0,Y 296.666,Z 397.141,A -85,B 0,C 180,E1 -16291.357,E2 -16291.357} C_VEL
LIN {X 0,Y 296.63,Z 396.663,A -85,B 0,C 180,E1 -16292.715,E2 -16292.715} C_VEL
LIN {X 0,Y 296.646,Z 395.746,A -85,B 0,C 180,E1 -16294.075,E2 -16294.075} C_VEL
LIN {X 0,Y 296.744,Z 393.919,A -85,B 0,C 180,E1 -16295.879,E2 -16295.879} C_VEL
LIN {X 0,Y 296.968,Z 390.524,A -85,B 0,C 180,E1 -16298.163,E2 -16298.163} C_VEL
LIN {X 0,Y 297.461,Z 386.383,A -85,B 0,C 180,E1 -16300.206,E2 -16300.206} C_VEL
LIN {X 0,Y 298.395,Z 380.076,A -85,B 0,C 180,E1 -16302.583,E2 -16302.583} C_VEL
LIN {X 0,Y 299.66,Z 373.262,A -85,B 0,C 180,E1 -16304.602,E2 -16304.602} C_VEL
LIN {X 0,Y 301.103,Z 365.184,A -85,B 0,C 180,E1 -16306.54,E2 -16306.54} C_VEL
LIN {X 0,Y 302.531,Z 356.343,A -85,B 0,C 180,E1 -16308.276,E2 -16308.276} C_VEL
LIN {X 0,Y 304.412,Z 345.92,A -85,B 0,C 180,E1 -16309.909,E2 -16309.909} C_VEL
LIN {X 0,Y 305.549,Z 338.517,A -85,B 0,C 180,E1 -16310.886,E2 -16310.886} C_VEL
LIN {X 0,Y 305.278,Z 326.436,A -85,B 0,C 180,E1 -16312.34,E2 -16312.34} C_VEL
LIN {X 0,Y 304.368,Z 314.844,A -85,B 0,C 180,E1 -16313.515,E2 -16313.515} C_VEL
LIN {X 0,Y 302.205,Z 302.095,A -85,B 0,C 180,E1 -16314.655,E2 -16314.655} C_VEL
LIN {X 0,Y 298.755,Z 288.465,A -85,B 0,C 180,E1 -16315.708,E2 -16315.708} C_VEL
LIN {X 0,Y 298.711,Z 287.903,A -85,B 0,C 180,E1 -16315.738,E2 -16315.738} C_VEL
LIN {X 0,Y 299.678,Z 281.321,A -85,B 0,C 180,E1 -16319.802,E2 -16319.802} C_VEL
LIN {X 0,Y 300.586,Z 275.871,A -85,B 0,C 180,E1 -16323.328,E2 -16323.328} C_VEL
LIN {X 0,Y 301.443,Z 271.243,A -85,B 0,C 180,E1 -16326.477,E2 -16326.477} C_VEL
LIN {X 0,Y 301.399,Z 267.847,A -85,B 0,C 180,E1 -16329.018,E2 -16329.018} C_VEL
LIN {X 0,Y 300.617,Z 263.429,A -85,B 0,C 180,E1 -16332.685,E2 -16332.685} C_VEL
LIN {X 0,Y 299.831,Z 259.197,A -85,B 0,C 180,E1 -16336.604,E2 -16336.604} C_VEL
LIN {X 0,Y 299.466,Z 257.008,A -85,B 0,C 180,E1 -16338.917,E2 -16338.917} C_VEL
LIN {X 0,Y 298.824,Z 253.473,A -85,B 0,C 180,E1 -16343.094,E2 -16343.094} C_VEL
LIN {X 0,Y 298.492,Z 251.674,A -85,B 0,C 180,E1 -16345.59,E2 -16345.59} C_VEL
LIN {X 0,Y 298.396,Z 251.314,A -85,B 0,C 180,E1 -16348.789,E2 -16348.789} C_VEL
LIN {X 0,Y 298.463,Z 251.309,A -85,B 0,C 180,E1 -16351.902,E2 -16351.902} C_VEL
LIN {X 0,Y 298.485,Z 251.305,A -85,B 0,C 180,E1 -16354.922,E2 -16354.922} C_VEL
LIN {X 0,Y 298.449,Z 251.306,A -85,B 0,C 180,E1 -16359.313,E2 -16359.313} C_VEL
LIN {X 0,Y 298.537,Z 251.294,A -85,B 0,C 180,E1 -16362.177,E2 -16362.177} C_VEL
LIN {X 0,Y 298.592,Z 251.289,A -85,B 0,C 180,E1 -16364.993,E2 -16364.993} C_VEL
LIN {X 0,Y 298.591,Z 251.288,A -85,B 0,C 180,E1 -16369.144,E2 -16369.144} C_VEL
LIN {X 0,Y 298.756,Z 251.269,A -85,B 0,C 180,E1 -16371.884,E2 -16371.884} C_VEL
LIN {X 0,Y 298.658,Z 251.285,A -85,B 0,C 180,E1 -16374.597,E2 -16374.597} C_VEL
LIN {X 0,Y 298.922,Z 251.252,A -85,B 0,C 180,E1 -16378.651,E2 -16378.651} C_VEL
LIN {X 0,Y 298.921,Z 251.25,A -85,B 0,C 180,E1 -16381.345,E2 -16381.345} C_VEL
LIN {X 0,Y 298.826,Z 251.549,A -85,B 0,C 180,E1 -16386.688,E2 -16386.688} C_VEL
LIN {X 0,Y 298.888,Z 253.043,A -85,B 0,C 180,E1 -16389.471,E2 -16389.471} C_VEL
LIN {X 0,Y 298.815,Z 254.669,A -85,B 0,C 180,E1 -16392.218,E2 -16392.218} C_VEL
LIN {X 0,Y 298.63,Z 256.573,A -85,B 0,C 180,E1 -16395.23,E2 -16395.23} C_VEL
LIN {X 0,Y 298.281,Z 259.493,A -85,B 0,C 180,E1 -16399.533,E2 -16399.533} C_VEL
LIN {X 0,Y 298.135,Z 260.758,A -85,B 0,C 180,E1 -16401.293,E2 -16401.293} C_VEL
LIN {X 0,Y 299.206,Z 263.757,A -85,B 0,C 180,E1 -16401.574,E2 -16401.574} C_VEL
LIN {X 0,Y 303.567,Z 275.053,A -85,B 0,C 180,E1 -16402.728,E2 -16402.728} C_VEL
LIN {X 0,Y 306.969,Z 286.829,A -85,B 0,C 180,E1 -16404.037,E2 -16404.037} C_VEL
LIN {X 0,Y 308.711,Z 295.446,A -85,B 0,C 180,E1 -16405.085,E2 -16405.085} C_VEL
LIN {X 0,Y 308.559,Z 298.84,A -85,B 0,C 180,E1 -16405.459,E2 -16405.459} C_VEL
LIN {X 0,Y 306.988,Z 309.862,A -85,B 0,C 180,E1 -16406.77,E2 -16406.77} C_VEL
LIN {X 0,Y 305.434,Z 319.183,A -85,B 0,C 180,E1 -16408.142,E2 -16408.142} C_VEL
LIN {X 0,Y 303.747,Z 328.452,A -85,B 0,C 180,E1 -16409.829,E2 -16409.829} C_VEL
LIN {X 0,Y 302.245,Z 336.138,A -85,B 0,C 180,E1 -16411.552,E2 -16411.552} C_VEL
LIN {X 0,Y 300.845,Z 343.019,A -85,B 0,C 180,E1 -16413.45,E2 -16413.45} C_VEL
LIN {X 0,Y 299.627,Z 348.633,A -85,B 0,C 180,E1 -16415.367,E2 -16415.367} C_VEL
LIN {X 0,Y 298.515,Z 354.008,A -85,B 0,C 180,E1 -16417.74,E2 -16417.74} C_VEL
LIN {X 0,Y 297.859,Z 357.077,A -85,B 0,C 180,E1 -16419.57,E2 -16419.57} C_VEL
LIN {X 0,Y 297.346,Z 359.373,A -85,B 0,C 180,E1 -16421.434,E2 -16421.434} C_VEL
LIN {X 0,Y 296.945,Z 360.911,A -85,B 0,C 180,E1 -16423.339,E2 -16423.339} C_VEL
LIN {X 0,Y 296.721,Z 361.662,A -85,B 0,C 180,E1 -16425.277,E2 -16425.277} C_VEL
LIN {X 0,Y 296.57,Z 361.563,A -85,B 0,C 180,E1 -16427.271,E2 -16427.271} C_VEL
LIN {X 0,Y 296.676,Z 360.572,A -85,B 0,C 180,E1 -16429.288,E2 -16429.288} C_VEL
